# B&R Automation Studio project NAELD004C00R10L518F00 (part 35)

#### Act_Main.st
```iecst
(** 2020-03-16 **)
ACTION Act_Main:

	IF bModuleNotOK = FALSE THEN
		CASE eStat OF

			LifterActIdle:
				IF eStatus <> Idle THEN	//Reset Data
					//Private
					fbStop(bEn := FALSE);
					fbRstAxisErr(bEn := FALSE);
					fbJog(bEn := FALSE);
					fbMovRel(bEn := FALSE);
					fbMovAbs(bEn := FALSE);
					fbHoming(bEn := FALSE);
					fbPwrOff(bEn := FALSE);
					fbPwrOn(bEn := FALSE);
					fbFullHm(bEn := FALSE);
					fbFullMovAbs(bEn := FALSE);
					fbFullMovRel(bEn := FALSE);
					fbSDOWrite(bEn := FALSE);
					fbTm(IN := FALSE);
					usiStep	:= 0;
					usiCount			:= 0;
					bNotInterruptible	:= FALSE;

					sStatTxt	:= a_sStatText[eStat];

				END_IF

				eStatus	:= Idle;

				IF EDGENEG(p_bManual) THEN
					fMotionCANRstCtrlWord(ADR(tyParamOutDriver));
				END_IF

			LifterActGoAPos:
				IF (eStatus = Idle OR eStatus = Busy) THEN

					eStatus	:= Busy;

					sStatTxt	:= a_sStatText[eStat];

					bNotInterruptible	:= TRUE;

					CASE usiStep OF
						0:	//Wait For Motion Parameter Update
							p_diMovePosInUM	:= p_diAPos;
							usiStep	:= 1;

						1:	//Check Position Difference
							IF tyParamOut.bPosDiff = TRUE THEN
								usiStep	:= 2;
							ELSE
								eStatus	:= Done;
							END_IF

						2:	//Move
							fbFullMovAbs.tyParamInDriver					:= tyParamInDriver;
							fbFullMovAbs.tyParamInMove.diPosInUM			:= p_diMovePosInUM;
							fbFullMovAbs.tyParamInMove.diDistInUM			:= p_diMoveDistInUM;
							fbFullMovAbs.tyParamInMove.diVelInUMPS			:= p_diMoveVelInUMPS;
							fbFullMovAbs.tyParamInMove.diAcc				:= p_diMoveAcc;
							fbFullMovAbs.tyParamInMove.diDec				:= p_diMoveDec;
							fbFullMovAbs.tyParamOut							:= tyParamOut;
							fbFullMovAbs(bEn := TRUE);

							IF fbFullMovAbs.udiStatus = 0 THEN
								eStatus	:= Done;
							ELSIF fbFullMovAbs.udiStatus < 65534 THEN
								eStatus		:= Error;

								IF fbFullMovAbs.udiStatus = 1401 THEN
									udiStatus	:= 10002;	//Power On Time Out While Going A Position
								ELSIF fbFullMovAbs.udiStatus = 1402 THEN
									udiStatus	:= 10003;	//Homing Time Out While Going A Position
								ELSIF fbFullMovAbs.udiStatus = 1403 THEN
									udiStatus	:= 10004;	//Move Absolute Time Out While Going A Position
								ELSIF fbFullMovAbs.udiStatus = 1405 THEN
									udiStatus	:= 10005;	//Stop Motion Time Out While Going A Position
								ELSIF fbFullMovAbs.udiStatus = 1408 THEN
									udiStatus	:= 10006;	//Axis Error Reset Failed While Going A Position
								ELSIF fbFullMovAbs.udiStatus = 1409 THEN
									udiStatus	:= 10007;	//Axis Error Occur In Move Absolute While Going A Position
								ELSIF fbFullMovAbs.udiStatus = 1411 THEN
									udiStatus	:= 10008;	//Axis Error Occur In Homing While Going A Position
								ELSIF fbFullMovAbs.udiStatus = 1412 THEN
									udiStatus	:= 10009;	//Homing Done But Home Flag Is Not Activated While Going A Position
								ELSIF fbFullMovAbs.udiStatus = 1413 THEN
									udiStatus	:= 10010;	//Forward Limit Activated In Homing While Going A Position
								ELSIF fbFullMovAbs.udiStatus = 1414 THEN
									udiStatus	:= 10011;	//Reverse Limit Activated In Homing While Going A Position
								ELSIF fbFullMovAbs.udiStatus = 1415 THEN
									udiStatus	:= 10012;	//Forward Limit Activated In Move Absolute While Going A Position
								ELSIF fbFullMovAbs.udiStatus = 1416 THEN
									udiStatus	:= 10013;	//Reverse Limit Activated In Move Absolute While Going A Position
								ELSE
									udiStatus	:= fbFullMovAbs.udiStatus;
								END_IF
							END_IF

					END_CASE

				END_IF

			LifterActGoBPos:
				IF (eStatus = Idle OR eStatus = Busy) THEN

					eStatus	:= Busy;

					sStatTxt	:= a_sStatText[eStat];

					bNotInterruptible	:= TRUE;

					CASE usiStep OF
						0:	//Wait For Motion Parameter Update
							p_diMovePosInUM	:= p_diBPos;
							usiStep	:= 1;

						1:	//Check Position Difference
							IF tyParamOut.bPosDiff = TRUE THEN
								usiStep	:= 2;
							ELSE
								eStatus	:= Done;
							END_IF

						2:	//Move
							fbFullMovAbs.tyParamInDriver					:= tyParamInDriver;
							fbFullMovAbs.tyParamInMove.diPosInUM			:= p_diMovePosInUM;
							fbFullMovAbs.tyParamInMove.diDistInUM			:= p_diMoveDistInUM;
							fbFullMovAbs.tyParamInMove.diVelInUMPS			:= p_diMoveVelInUMPS;
							fbFullMovAbs.tyParamInMove.diAcc				:= p_diMoveAcc;
							fbFullMovAbs.tyParamInMove.diDec				:= p_diMoveDec;
							fbFullMovAbs.tyParamOut							:= tyParamOut;
							fbFullMovAbs(bEn := TRUE);

							IF fbFullMovAbs.udiStatus = 0 THEN
								eStatus	:= Done;
							ELSIF fbFullMovAbs.udiStatus < 65534 THEN
								eStatus		:= Error;

								IF fbFullMovAbs.udiStatus = 1401 THEN
									udiStatus	:= 10029;	//Power On Time Out While Going B Position
								ELSIF fbFullMovAbs.udiStatus = 1402 THEN
									udiStatus	:= 10030;	//Homing Time Out While Going B Position
								ELSIF fbFullMovAbs.udiStatus = 1403 THEN
									udiStatus	:= 10031;	//Move Absolute Time Out While Going B Position
								ELSIF fbFullMovAbs.udiStatus = 1405 THEN
									udiStatus	:= 10032;	//Stop Motion Time Out While Going B Position
								ELSIF fbFullMovAbs.udiStatus = 1408 THEN
									udiStatus	:= 10033;	//Axis Error Reset Failed While Going B Position
								ELSIF fbFullMovAbs.udiStatus = 1409 THEN
									udiStatus	:= 10034;	//Axis Error Occur In Move Absolute While Going B Position
								ELSIF fbFullMovAbs.udiStatus = 1411 THEN
									udiStatus	:= 10035;	//Axis Error Occur In Homing While Going B Position
								ELSIF fbFullMovAbs.udiStatus = 1412 THEN
									udiStatus	:= 10036;	//Homing Done But Home Flag Is Not Activated While Going B Position
								ELSIF fbFullMovAbs.udiStatus = 1413 THEN
									udiStatus	:= 10037;	//Forward Limit Activated In Homing While Going B Position
								ELSIF fbFullMovAbs.udiStatus = 1414 THEN
									udiStatus	:= 10038;	//Reverse Limit Activated In Homing While Going B Position
								ELSIF fbFullMovAbs.udiStatus = 1415 THEN
									udiStatus	:= 10039;	//Forward Limit Activated In Move Absolute While Going B Position
								ELSIF fbFullMovAbs.udiStatus = 1416 THEN
									udiStatus	:= 10040;	//Reverse Limit Activated In Move Absolute While Going B Position
								ELSE
									udiStatus	:= fbFullMovAbs.udiStatus;
								END_IF
							END_IF

					END_CASE

				END_IF

			LifterActGoCPos:
				IF (eStatus = Idle OR eStatus = Busy) THEN

					eStatus	:= Busy;

					sStatTxt	:= a_sStatText[eStat];

					bNotInterruptible	:= TRUE;

					CASE usiStep OF
						0:	//Wait For Motion Parameter Update
							p_diMovePosInUM	:= p_diCPos;
							usiStep	:= 1;

						1:	//Check Position Difference
							IF tyParamOut.bPosDiff = TRUE THEN
								usiStep	:= 2;
							ELSE
								eStatus	:= Done;
							END_IF

						2:	//Move
							fbFullMovAbs.tyParamInDriver					:= tyParamInDriver;
							fbFullMovAbs.tyParamInMove.diPosInUM			:= p_diMovePosInUM;
							fbFullMovAbs.tyParamInMove.diDistInUM			:= p_diMoveDistInUM;
							fbFullMovAbs.tyParamInMove.diVelInUMPS			:= p_diMoveVelInUMPS;
							fbFullMovAbs.tyParamInMove.diAcc				:= p_diMoveAcc;
							fbFullMovAbs.tyParamInMove.diDec				:= p_diMoveDec;
							fbFullMovAbs.tyParamOut							:= tyParamOut;
							fbFullMovAbs(bEn := TRUE);

							IF fbFullMovAbs.udiStatus = 0 THEN
								eStatus	:= Done;
							ELSIF fbFullMovAbs.udiStatus < 65534 THEN
								eStatus		:= Error;

								IF fbFullMovAbs.udiStatus = 1401 THEN
									udiStatus	:= 10078;	//Power On Time Out While Going C Position
								ELSIF fbFullMovAbs.udiStatus = 1402 THEN
									udiStatus	:= 10079;	//Homing Time Out While Going C Position
								ELSIF fbFullMovAbs.udiStatus = 1403 THEN
									udiStatus	:= 10080;	//Move Absolute Time Out While Going C Position
								ELSIF fbFullMovAbs.udiStatus = 1405 THEN
									udiStatus	:= 10081;	//Stop Motion Time Out While Going C Position
								ELSIF fbFullMovAbs.udiStatus = 1408 THEN
									udiStatus	:= 10082;	//Axis Error Reset Failed While Going C Position
								ELSIF fbFullMovAbs.udiStatus = 1409 THEN
									udiStatus	:= 10083;	//Axis Error Occur In Move Absolute While Going C Position
								ELSIF fbFullMovAbs.udiStatus = 1411 THEN
									udiStatus	:= 10084;	//Axis Error Occur In Homing While Going C Position
								ELSIF fbFullMovAbs.udiStatus = 1412 THEN
									udiStatus	:= 10085;	//Homing Done But Home Flag Is Not Activated While Going C Position
								ELSIF fbFullMovAbs.udiStatus = 1413 THEN
									udiStatus	:= 10086;	//Forward Limit Activated In Homing While Going C Position
								ELSIF fbFullMovAbs.udiStatus = 1414 THEN
									udiStatus	:= 10087;	//Reverse Limit Activated In Homing While Going C Position
								ELSIF fbFullMovAbs.udiStatus = 1415 THEN
									udiStatus	:= 10088;	//Forward Limit Activated In Move Absolute While Going C Position
								ELSIF fbFullMovAbs.udiStatus = 1416 THEN
									udiStatus	:= 10089;	//Reverse Limit Activated In Move Absolute While Going C Position
								ELSE
									udiStatus	:= fbFullMovAbs.udiStatus;
								END_IF
							END_IF

					END_CASE

				END_IF

			LifterActGoDPos:
				IF (eStatus = Idle OR eStatus = Busy) THEN

					eStatus	:= Busy;

					sStatTxt	:= a_sStatText[eStat];

					bNotInterruptible	:= TRUE;

					CASE usiStep OF
						0:	//Wait For Motion Parameter Update
							p_diMovePosInUM	:= p_diDPos;
							usiStep	:= 1;

						1:	//Check Position Difference
							IF tyParamOut.bPosDiff = TRUE THEN
								usiStep	:= 2;
							ELSE
								eStatus	:= Done;
							END_IF

						2:	//Move
							fbFullMovAbs.tyParamInDriver					:= tyParamInDriver;
							fbFullMovAbs.tyParamInMove.diPosInUM			:= p_diMovePosInUM;
							fbFullMovAbs.tyParamInMove.diDistInUM			:= p_diMoveDistInUM;
							fbFullMovAbs.tyParamInMove.diVelInUMPS			:= p_diMoveVelInUMPS;
							fbFullMovAbs.tyParamInMove.diAcc				:= p_diMoveAcc;
							fbFullMovAbs.tyParamInMove.diDec				:= p_diMoveDec;
							fbFullMovAbs.tyParamOut							:= tyParamOut;
							fbFullMovAbs(bEn := TRUE);

							IF fbFullMovAbs.udiStatus = 0 THEN
								eStatus	:= Done;
							ELSIF fbFullMovAbs.udiStatus < 65534 THEN
								eStatus		:= Error;

								IF fbFullMovAbs.udiStatus = 1401 THEN
									udiStatus	:= 10090;	//Power On Time Out While Going D Position
								ELSIF fbFullMovAbs.udiStatus = 1402 THEN
									udiStatus	:= 10091;	//Homing Time Out While Going D Position
								ELSIF fbFullMovAbs.udiStatus = 1403 THEN
									udiStatus	:= 10092;	//Move Absolute Time Out While Going D Position
								ELSIF fbFullMovAbs.udiStatus = 1405 THEN
									udiStatus	:= 10093;	//Stop Motion Time Out While Going D Position
								ELSIF fbFullMovAbs.udiStatus = 1408 THEN
									udiStatus	:= 10094;	//Axis Error Reset Failed While Going D Position
								ELSIF fbFullMovAbs.udiStatus = 1409 THEN
									udiStatus	:= 10095;	//Axis Error Occur In Move Absolute While Going D Position
								ELSIF fbFullMovAbs.udiStatus = 1411 THEN
									udiStatus	:= 10096;	//Axis Error Occur In Homing While Going D Position
								ELSIF fbFullMovAbs.udiStatus = 1412 THEN
									udiStatus	:= 10097;	//Homing Done But Home Flag Is Not Activated While Going D Position
								ELSIF fbFullMovAbs.udiStatus = 1413 THEN
									udiStatus	:= 10098;	//Forward Limit Activated In Homing While Going D Position
								ELSIF fbFullMovAbs.udiStatus = 1414 THEN
									udiStatus	:= 10099;	//Reverse Limit Activated In Homing While Going D Position
								ELSIF fbFullMovAbs.udiStatus = 1415 THEN
									udiStatus	:= 10100;	//Forward Limit Activated In Move Absolute While Going D Position
								ELSIF fbFullMovAbs.udiStatus = 1416 THEN
									udiStatus	:= 10101;	//Reverse Limit Activated In Move Absolute While Going D Position
								ELSE
									udiStatus	:= fbFullMovAbs.udiStatus;
								END_IF
							END_IF

					END_CASE

				END_IF

			LifterActGoEPos:
				IF (eStatus = Idle OR eStatus = Busy) THEN

					eStatus	:= Busy;

					sStatTxt	:= a_sStatText[eStat];

					bNotInterruptible	:= TRUE;

					CASE usiStep OF
						0:	//Wait For Motion Parameter Update
							p_diMovePosInUM	:= p_diEPos;
							usiStep	:= 1;

						1:	//Check Position Difference
							IF tyParamOut.bPosDiff = TRUE THEN
								usiStep	:= 2;
							ELSE
								eStatus	:= Done;
							END_IF

						2:	//Move
							fbFullMovAbs.tyParamInDriver					:= tyParamInDriver;
							fbFullMovAbs.tyParamInMove.diPosInUM			:= p_diMovePosInUM;
							fbFullMovAbs.tyParamInMove.diDistInUM			:= p_diMoveDistInUM;
							fbFullMovAbs.tyParamInMove.diVelInUMPS			:= p_diMoveVelInUMPS;
							fbFullMovAbs.tyParamInMove.diAcc				:= p_diMoveAcc;
							fbFullMovAbs.tyParamInMove.diDec				:= p_diMoveDec;
							fbFullMovAbs.tyParamOut							:= tyParamOut;
							fbFullMovAbs(bEn := TRUE);

							IF fbFullMovAbs.udiStatus = 0 THEN
								eStatus	:= Done;
							ELSIF fbFullMovAbs.udiStatus < 65534 THEN
								eStatus		:= Error;

								IF fbFullMovAbs.udiStatus = 1401 THEN
									udiStatus	:= 10102;	//Power On Time Out While Going E Position
								ELSIF fbFullMovAbs.udiStatus = 1402 THEN
									udiStatus	:= 10103;	//Homing Time Out While Going E Position
								ELSIF fbFullMovAbs.udiStatus = 1403 THEN
									udiStatus	:= 10104;	//Move Absolute Time Out While Going E Position
								ELSIF fbFullMovAbs.udiStatus = 1405 THEN
									udiStatus	:= 10105;	//Stop Motion Time Out While Going E Position
								ELSIF fbFullMovAbs.udiStatus = 1408 THEN
									udiStatus	:= 10106;	//Axis Error Reset Failed While Going E Position
								ELSIF fbFullMovAbs.udiStatus = 1409 THEN
									udiStatus	:= 10107;	//Axis Error Occur In Move Absolute While Going E Position
								ELSIF fbFullMovAbs.udiStatus = 1411 THEN
									udiStatus	:= 10108;	//Axis Error Occur In Homing While Going E Position
								ELSIF fbFullMovAbs.udiStatus = 1412 THEN
									udiStatus	:= 10109;	//Homing Done But Home Flag Is Not Activated While Going E Position
								ELSIF fbFullMovAbs.udiStatus = 1413 THEN
									udiStatus	:= 10110;	//Forward Limit Activated In Homing While Going E Position
								ELSIF fbFullMovAbs.udiStatus = 1414 THEN
									udiStatus	:= 10111;	//Reverse Limit Activated In Homing While Going E Position
								ELSIF fbFullMovAbs.udiStatus = 1415 THEN
									udiStatus	:= 10112;	//Forward Limit Activated In Move Absolute While Going E Position
								ELSIF fbFullMovAbs.udiStatus = 1416 THEN
									udiStatus	:= 10113;	//Reverse Limit Activated In Move Absolute While Going E Position
								ELSE
									udiStatus	:= fbFullMovAbs.udiStatus;
								END_IF
							END_IF

					END_CASE

				END_IF

			LifterActGoFPos:
				IF (eStatus = Idle OR eStatus = Busy) THEN

					eStatus	:= Busy;

					sStatTxt	:= a_sStatText[eStat];

					bNotInterruptible	:= TRUE;

					CASE usiStep OF
						0:	//Wait For Motion Parameter Update
							p_diMovePosInUM	:= p_diFPos;
							usiStep	:= 1;

						1:	//Check Position Difference
							IF tyParamOut.bPosDiff = TRUE THEN
								usiStep	:= 2;
							ELSE
								eStatus	:= Done;
							END_IF

						2:	//Move
							fbFullMovAbs.tyParamInDriver					:= tyParamInDriver;
							fbFullMovAbs.tyParamInMove.diPosInUM			:= p_diMovePosInUM;
							fbFullMovAbs.tyParamInMove.diDistInUM			:= p_diMoveDistInUM;
							fbFullMovAbs.tyParamInMove.diVelInUMPS			:= p_diMoveVelInUMPS;
							fbFullMovAbs.tyParamInMove.diAcc				:= p_diMoveAcc;
							fbFullMovAbs.tyParamInMove.diDec				:= p_diMoveDec;
							fbFullMovAbs.tyParamOut							:= tyParamOut;
							fbFullMovAbs(bEn := TRUE);

							IF fbFullMovAbs.udiStatus = 0 THEN
								eStatus	:= Done;
							ELSIF fbFullMovAbs.udiStatus < 65534 THEN
								eStatus		:= Error;

								IF fbFullMovAbs.udiStatus = 1401 THEN
									udiStatus	:= 10114;	//Power On Time Out While Going F Position
								ELSIF fbFullMovAbs.udiStatus = 1402 THEN
									udiStatus	:= 10115;	//Homing Time Out While Going F Position
								ELSIF fbFullMovAbs.udiStatus = 1403 THEN
									udiStatus	:= 10116;	//Move Absolute Time Out While Going F Position
								ELSIF fbFullMovAbs.udiStatus = 1405 THEN
									udiStatus	:= 10117;	//Stop Motion Time Out While Going F Position
								ELSIF fbFullMovAbs.udiStatus = 1408 THEN
									udiStatus	:= 10118;	//Axis Error Reset Failed While Going F Position
								ELSIF fbFullMovAbs.udiStatus = 1409 THEN
									udiStatus	:= 10119;	//Axis Error Occur In Move Absolute While Going F Position
								ELSIF fbFullMovAbs.udiStatus = 1411 THEN
									udiStatus	:= 10120;	//Axis Error Occur In Homing While Going F Position
								ELSIF fbFullMovAbs.udiStatus = 1412 THEN
									udiStatus	:= 10121;	//Homing Done But Home Flag Is Not Activated While Going F Position
								ELSIF fbFullMovAbs.udiStatus = 1413 THEN
									udiStatus	:= 10122;	//Forward Limit Activated In Homing While Going F Position
								ELSIF fbFullMovAbs.udiStatus = 1414 THEN
									udiStatus	:= 10123;	//Reverse Limit Activated In Homing While Going F Position
								ELSIF fbFullMovAbs.udiStatus = 1415 THEN
									udiStatus	:= 10124;	//Forward Limit Activated In Move Absolute While Going F Position
								ELSIF fbFullMovAbs.udiStatus = 1416 THEN
									udiStatus	:= 10125;	//Reverse Limit Activated In Move Absolute While Going F Position
								ELSE
									udiStatus	:= fbFullMovAbs.udiStatus;
								END_IF
							END_IF

					END_CASE

				END_IF

			LifterActGoGPos:
				IF (eStatus = Idle OR eStatus = Busy) THEN

					eStatus	:= Busy;

					sStatTxt	:= a_sStatText[eStat];

					bNotInterruptible	:= TRUE;

					CASE usiStep OF
						0:	//Wait For Motion Parameter Update
							p_diMovePosInUM	:= p_diGPos;
							usiStep	:= 1;

						1:	//Check Position Difference
							IF tyParamOut.bPosDiff = TRUE THEN
								usiStep	:= 2;
							ELSE
								eStatus	:= Done;
							END_IF

						2:	//Move
							fbFullMovAbs.tyParamInDriver					:= tyParamInDriver;
							fbFullMovAbs.tyParamInMove.diPosInUM			:= p_diMovePosInUM;
							fbFullMovAbs.tyParamInMove.diDistInUM			:= p_diMoveDistInUM;
							fbFullMovAbs.tyParamInMove.diVelInUMPS			:= p_diMoveVelInUMPS;
							fbFullMovAbs.tyParamInMove.diAcc				:= p_diMoveAcc;
							fbFullMovAbs.tyParamInMove.diDec				:= p_diMoveDec;
							fbFullMovAbs.tyParamOut							:= tyParamOut;
							fbFullMovAbs(bEn := TRUE);

							IF fbFullMovAbs.udiStatus = 0 THEN
								eStatus	:= Done;
							ELSIF fbFullMovAbs.udiStatus < 65534 THEN
								eStatus		:= Error;

								IF fbFullMovAbs.udiStatus = 1401 THEN
									udiStatus	:= 10126;	//Power On Time Out While Going G Position
								ELSIF fbFullMovAbs.udiStatus = 1402 THEN
									udiStatus	:= 10127;	//Homing Time Out While Going G Position
								ELSIF fbFullMovAbs.udiStatus = 1403 THEN
									udiStatus	:= 10128;	//Move Absolute Time Out While Going G Position
								ELSIF fbFullMovAbs.udiStatus = 1405 THEN
									udiStatus	:= 10129;	//Stop Motion Time Out While Going G Position
								ELSIF fbFullMovAbs.udiStatus = 1408 THEN
									udiStatus	:= 10130;	//Axis Error Reset Failed While Going G Position
								ELSIF fbFullMovAbs.udiStatus = 1409 THEN
									udiStatus	:= 10131;	//Axis Error Occur In Move Absolute While Going G Position
								ELSIF fbFullMovAbs.udiStatus = 1411 THEN
									udiStatus	:= 10132;	//Axis Error Occur In Homing While Going G Position
								ELSIF fbFullMovAbs.udiStatus = 1412 THEN
									udiStatus	:= 10133;	//Homing Done But Home Flag Is Not Activated While Going G Position
								ELSIF fbFullMovAbs.udiStatus = 1413 THEN
									udiStatus	:= 10134;	//Forward Limit Activated In Homing While Going G Position
								ELSIF fbFullMovAbs.udiStatus = 1414 THEN
									udiStatus	:= 10135;	//Reverse Limit Activated In Homing While Going G Position
								ELSIF fbFullMovAbs.udiStatus = 1415 THEN
									udiStatus	:= 10136;	//Forward Limit Activated In Move Absolute While Going G Position
								ELSIF fbFullMovAbs.udiStatus = 1416 THEN
									udiStatus	:= 10137;	//Reverse Limit Activated In Move Absolute While Going G Position
								ELSE
									udiStatus	:= fbFullMovAbs.udiStatus;
								END_IF
							END_IF

					END_CASE

				END_IF

			LifterActGoHPos:
				IF (eStatus = Idle OR eStatus = Busy) THEN

					eStatus	:= Busy;

					sStatTxt	:= a_sStatText[eStat];

					bNotInterruptible	:= TRUE;

					CASE usiStep OF
						0:	//Wait For Motion Parameter Update
							p_diMovePosInUM	:= p_diHPos;
							usiStep	:= 1;

						1:	//Check Position Difference
							IF tyParamOut.bPosDiff = TRUE THEN
								usiStep	:= 2;
							ELSE
								eStatus	:= Done;
							END_IF

						2:	//Move
							fbFullMovAbs.tyParamInDriver					:= tyParamInDriver;
							fbFullMovAbs.tyParamInMove.diPosInUM			:= p_diMovePosInUM;
							fbFullMovAbs.tyParamInMove.diDistInUM			:= p_diMoveDistInUM;
							fbFullMovAbs.tyParamInMove.diVelInUMPS			:= p_diMoveVelInUMPS;
							fbFullMovAbs.tyParamInMove.diAcc				:= p_diMoveAcc;
							fbFullMovAbs.tyParamInMove.diDec				:= p_diMoveDec;
							fbFullMovAbs.tyParamOut							:= tyParamOut;
							fbFullMovAbs(bEn := TRUE);

							IF fbFullMovAbs.udiStatus = 0 THEN
								eStatus	:= Done;
							ELSIF fbFullMovAbs.udiStatus < 65534 THEN
								eStatus		:= Error;

								IF fbFullMovAbs.udiStatus = 1401 THEN
									udiStatus	:= 10138;	//Power On Time Out While Going H Position
								ELSIF fbFullMovAbs.udiStatus = 1402 THEN
									udiStatus	:= 10139;	//Homing Time Out While Going H Position
								ELSIF fbFullMovAbs.udiStatus = 1403 THEN
									udiStatus	:= 10140;	//Move Absolute Time Out While Going H Position
								ELSIF fbFullMovAbs.udiStatus = 1405 THEN
									udiStatus	:= 10141;	//Stop Motion Time Out While Going H Position
								ELSIF fbFullMovAbs.udiStatus = 1408 THEN
									udiStatus	:= 10142;	//Axis Error Reset Failed While Going H Position
								ELSIF fbFullMovAbs.udiStatus = 1409 THEN
									udiStatus	:= 10143;	//Axis Error Occur In Move Absolute While Going H Position
								ELSIF fbFullMovAbs.udiStatus = 1411 THEN
									udiStatus	:= 10144;	//Axis Error Occur In Homing While Going H Position
								ELSIF fbFullMovAbs.udiStatus = 1412 THEN
									udiStatus	:= 10145;	//Homing Done But Home Flag Is Not Activated While Going H Position
								ELSIF fbFullMovAbs.udiStatus = 1413 THEN
									udiStatus	:= 10146;	//Forward Limit Activated In Homing While Going H Position
								ELSIF fbFullMovAbs.udiStatus = 1414 THEN
									udiStatus	:= 10147;	//Reverse Limit Activated In Homing While Going H Position
								ELSIF fbFullMovAbs.udiStatus = 1415 THEN
									udiStatus	:= 10148;	//Forward Limit Activated In Move Absolute While Going H Position
								ELSIF fbFullMovAbs.udiStatus = 1416 THEN
									udiStatus	:= 10149;	//Reverse Limit Activated In Move Absolute While Going H Position
								ELSE
									udiStatus	:= fbFullMovAbs.udiStatus;
								END_IF
							END_IF

					END_CASE

				END_IF

			LifterActGoASltPos:
				IF (eStatus = Idle OR eStatus = Busy) THEN

					eStatus	:= Busy;

					sStatTxt	:= a_sStatText[eStat];

					bNotInterruptible	:= TRUE;

					CASE usiStep OF
						0:	//Wait For Motion Parameter Update
							p_diMovePosInUM	:= fLifterSltToPosInUMBtmMin(p_diGoASlt , p_diASltToSltDist , p_diASlt1Pos);
							usiStep	:= 1;

						1:	//Check Position Difference
							IF tyParamOut.bPosDiff = TRUE THEN
								usiStep	:= 2;
							ELSE
								eStatus	:= Done;
							END_IF

						2:	//Move
							fbFullMovAbs.tyParamInDriver					:= tyParamInDriver;
							fbFullMovAbs.tyParamInMove.diPosInUM			:= p_diMovePosInUM;
							fbFullMovAbs.tyParamInMove.diDistInUM			:= p_diMoveDistInUM;
							fbFullMovAbs.tyParamInMove.diVelInUMPS			:= p_diMoveVelInUMPS;
							fbFullMovAbs.tyParamInMove.diAcc				:= p_diMoveAcc;
							fbFullMovAbs.tyParamInMove.diDec				:= p_diMoveDec;
							fbFullMovAbs.tyParamOut							:= tyParamOut;
							fbFullMovAbs(bEn := TRUE);

							IF fbFullMovAbs.udiStatus = 0 THEN
								eStatus	:= Done;
							ELSIF fbFullMovAbs.udiStatus < 65534 THEN
								eStatus		:= Error;

								IF fbFullMovAbs.udiStatus = 1401 THEN
									udiStatus	:= 10041;	//Power On Time Out While Going New A Slot Position
								ELSIF fbFullMovAbs.udiStatus = 1402 THEN
									udiStatus	:= 10042;	//Homing Time Out While Going New A Slot Position
								ELSIF fbFullMovAbs.udiStatus = 1403 THEN
									udiStatus	:= 10043;	//Move Absolute Time Out While Going New A Slot Position
								ELSIF fbFullMovAbs.udiStatus = 1405 THEN
									udiStatus	:= 10044;	//Stop Motion Time Out While Going New A Slot Position
								ELSIF fbFullMovAbs.udiStatus = 1408 THEN
									udiStatus	:= 10045;	//Axis Error Reset Failed While Going New A Slot Position
								ELSIF fbFullMovAbs.udiStatus = 1409 THEN
									udiStatus	:= 10046;	//Axis Error Occur In Move Absolute While Going New A Slot Position
								ELSIF fbFullMovAbs.udiStatus = 1411 THEN
									udiStatus	:= 10047;	//Axis Error Occur In Homing While Going New A Slot Position
								ELSIF fbFullMovAbs.udiStatus = 1412 THEN
									udiStatus	:= 10048;	//Homing Done But Home Flag Is Not Activated While Going New A Slot Position
								ELSIF fbFullMovAbs.udiStatus = 1413 THEN
									udiStatus	:= 10049;	//Forward Limit Activated In Homing While Going New A Slot Position
								ELSIF fbFullMovAbs.udiStatus = 1414 THEN
									udiStatus	:= 10050;	//Reverse Limit Activated In Homing While Going New A Slot Position
								ELSIF fbFullMovAbs.udiStatus = 1415 THEN
									udiStatus	:= 10051;	//Forward Limit Activated In Move Absolute While Going New A Slot Position
								ELSIF fbFullMovAbs.udiStatus = 1416 THEN
									udiStatus	:= 10052;	//Reverse Limit Activated In Move Absolute While Going New A Slot Position
								ELSE
									udiStatus	:= fbFullMovAbs.udiStatus;
								END_IF
							END_IF

					END_CASE

				END_IF

			LifterActGoNxtASltPos:
				IF (eStatus = Idle OR eStatus = Busy) THEN

					eStatus	:= Busy;

					sStatTxt	:= a_sStatText[eStat];

					bNotInterruptible	:= TRUE;

					CASE usiStep OF
						0:	//Wait For Motion Parameter Update
							diExpectSlt		:= fLifterPosInUMToSltBtmMin(tyParamOut.diActualPosInUM , p_diASltToSltDist , p_diASlt1Pos);
							diExpectPosInUM	:= fLifterSltToPosInUMBtmMin(diExpectSlt , p_diASltToSltDist , p_diASlt1Pos);

							IF ABS(tyParamOut.diActualPosInUM - diExpectPosInUM) < 50 THEN
								p_diGoASlt		:= diExpectSlt + 1;
								p_diMovePosInUM	:= fLifterSltToPosInUMBtmMin(p_diGoASlt , p_diASltToSltDist , p_diASlt1Pos);

							ELSIF tyParamOut.diActualPosInUM > diExpectPosInUM THEN
								p_diGoASlt		:= diExpectSlt;
								p_diMovePosInUM	:= fLifterSltToPosInUMBtmMin(p_diGoASlt , p_diASltToSltDist , p_diASlt1Pos);

							ELSIF tyParamOut.diActualPosInUM < diExpectPosInUM THEN
								p_diGoASlt		:= diExpectSlt + 1;
								p_diMovePosInUM	:= fLifterSltToPosInUMBtmMin(p_diGoASlt , p_diASltToSltDist , p_diASlt1Pos);

							END_IF

							usiStep	:= 1;

						1:	//Check Position Difference
							IF tyParamOut.bPosDiff = TRUE THEN
								usiStep	:= 2;
							ELSE
								eStatus	:= Done;
							END_IF

						2:	//Move
							fbFullMovAbs.tyParamInDriver					:= tyParamInDriver;
							fbFullMovAbs.tyParamInMove.diPosInUM			:= p_diMovePosInUM;
							fbFullMovAbs.tyParamInMove.diDistInUM			:= p_diMoveDistInUM;
							fbFullMovAbs.tyParamInMove.diVelInUMPS			:= p_diMoveVelInUMPS;
							fbFullMovAbs.tyParamInMove.diAcc				:= p_diMoveAcc;
							fbFullMovAbs.tyParamInMove.diDec				:= p_diMoveDec;
							fbFullMovAbs.tyParamOut							:= tyParamOut;
							fbFullMovAbs(bEn := TRUE);

							IF fbFullMovAbs.udiStatus = 0 THEN
								eStatus	:= Done;
							ELSIF fbFullMovAbs.udiStatus < 65534 THEN
								eStatus		:= Error;

								IF fbFullMovAbs.udiStatus = 1401 THEN
									udiStatus	:= 10053;	//Power On Time Out While Going Next A Slot Position
								ELSIF fbFullMovAbs.udiStatus = 1402 THEN
									udiStatus	:= 10054;	//Homing Time Out While Going Next A Slot Position
								ELSIF fbFullMovAbs.udiStatus = 1403 THEN
									udiStatus	:= 10055;	//Move Absolute Time Out While Going Next A Slot Position
								ELSIF fbFullMovAbs.udiStatus = 1405 THEN
									udiStatus	:= 10056;	//Stop Motion Time Out While Going Next A Slot Position
								ELSIF fbFullMovAbs.udiStatus = 1408 THEN
									udiStatus	:= 10057;	//Axis Error Reset Failed While Going Next A Slot Position
								ELSIF fbFullMovAbs.udiStatus = 1409 THEN
									udiStatus	:= 10058;	//Axis Error Occur In Move Absolute While Going Next A Slot Position
								ELSIF fbFullMovAbs.udiStatus = 1411 THEN
									udiStatus	:= 10059;	//Axis Error Occur In Homing While Going Next A Slot Position
								ELSIF fbFullMovAbs.udiStatus = 1412 THEN
									udiStatus	:= 10060;	//Homing Done But Home Flag Is Not Activated While Going Next A Slot Position
								ELSIF fbFullMovAbs.udiStatus = 1413 THEN
									udiStatus	:= 10061;	//Forward Limit Activated In Homing While Going Next A Slot Position
								ELSIF fbFullMovAbs.udiStatus = 1414 THEN
									udiStatus	:= 10062;	//Reverse Limit Activated In Homing While Going Next A Slot Position
								ELSIF fbFullMovAbs.udiStatus = 1415 THEN
									udiStatus	:= 10063;	//Forward Limit Activated In Move Absolute While Going Next A Slot Position
								ELSIF fbFullMovAbs.udiStatus = 1416 THEN
									udiStatus	:= 10064;	//Reverse Limit Activated In Move Absolute While Going Next A Slot Position
								ELSE
									udiStatus	:= fbFullMovAbs.udiStatus;
								END_IF
							END_IF

					END_CASE

				END_IF

			LifterActGoPrevASltPos:
				IF (eStatus = Idle OR eStatus = Busy) THEN

					eStatus	:= Busy;

					sStatTxt	:= a_sStatText[eStat];

					bNotInterruptible	:= TRUE;

					CASE usiStep OF
						0:	//Wait For Motion Parameter Update
							diExpectSlt		:= fLifterPosInUMToSltBtmMin(tyParamOut.diActualPosInUM , p_diASltToSltDist , p_diASlt1Pos);
							diExpectPosInUM	:= fLifterSltToPosInUMBtmMin(diExpectSlt , p_diASltToSltDist , p_diASlt1Pos);

							IF ABS(tyParamOut.diActualPosInUM - diExpectPosInUM) < 50 THEN
								p_diGoASlt		:= diExpectSlt - 1;
								p_diMovePosInUM	:= fLifterSltToPosInUMBtmMin(p_diGoASlt , p_diASltToSltDist , p_diASlt1Pos);

							ELSIF tyParamOut.diActualPosInUM > diExpectPosInUM THEN
								p_diGoASlt		:= diExpectSlt - 1;
								p_diMovePosInUM	:= fLifterSltToPosInUMBtmMin(p_diGoASlt , p_diASltToSltDist , p_diASlt1Pos);

							ELSIF tyParamOut.diActualPosInUM < diExpectPosInUM THEN
								p_diGoASlt		:= diExpectSlt;
								p_diMovePosInUM	:= fLifterSltToPosInUMBtmMin(p_diGoASlt , p_diASltToSltDist , p_diASlt1Pos);

							END_IF

							usiStep	:= 1;

						1:	//Check Position Difference
							IF tyParamOut.bPosDiff = TRUE THEN
								usiStep	:= 2;
							ELSE
								eStatus	:= Done;
							END_IF

						2:	//Move
							fbFullMovAbs.tyParamInDriver					:= tyParamInDriver;
							fbFullMovAbs.tyParamInMove.diPosInUM			:= p_diMovePosInUM;
							fbFullMovAbs.tyParamInMove.diDistInUM			:= p_diMoveDistInUM;
							fbFullMovAbs.tyParamInMove.diVelInUMPS			:= p_diMoveVelInUMPS;
							fbFullMovAbs.tyParamInMove.diAcc				:= p_diMoveAcc;
							fbFullMovAbs.tyParamInMove.diDec				:= p_diMoveDec;
							fbFullMovAbs.tyParamOut							:= tyParamOut;
							fbFullMovAbs(bEn := TRUE);

							IF fbFullMovAbs.udiStatus = 0 THEN
								eStatus	:= Done;
							ELSIF fbFullMovAbs.udiStatus < 65534 THEN
								eStatus		:= Error;

								IF fbFullMovAbs.udiStatus = 1401 THEN
									udiStatus	:= 10065;	//Power On Time Out While Going Previous A Slot Position
								ELSIF fbFullMovAbs.udiStatus = 1402 THEN
									udiStatus	:= 10066;	//Homing Time Out While Going Previous A Slot Position
								ELSIF fbFullMovAbs.udiStatus = 1403 THEN
									udiStatus	:= 10067;	//Move Absolute Time Out While Going Previous A Slot Position
								ELSIF fbFullMovAbs.udiStatus = 1405 THEN
									udiStatus	:= 10068;	//Stop Motion Time Out While Going Previous A Slot Position
								ELSIF fbFullMovAbs.udiStatus = 1408 THEN
									udiStatus	:= 10069;	//Axis Error Reset Failed While Going Previous A Slot Position
								ELSIF fbFullMovAbs.udiStatus = 1409 THEN
									udiStatus	:= 10070;	//Axis Error Occur In Move Absolute While Going Previous A Slot Position
								ELSIF fbFullMovAbs.udiStatus = 1411 THEN
									udiStatus	:= 10071;	//Axis Error Occur In Homing While Going Previous A Slot Position
								ELSIF fbFullMovAbs.udiStatus = 1412 THEN
									udiStatus	:= 10072;	//Homing Done But Home Flag Is Not Activated While Going Previous A Slot Position
								ELSIF fbFullMovAbs.udiStatus = 1413 THEN
									udiStatus	:= 10073;	//Forward Limit Activated In Homing While Going Previous A Slot Position
								ELSIF fbFullMovAbs.udiStatus = 1414 THEN
									udiStatus	:= 10074;	//Reverse Limit Activated In Homing While Going Previous A Slot Position
								ELSIF fbFullMovAbs.udiStatus = 1415 THEN
									udiStatus	:= 10075;	//Forward Limit Activated In Move Absolute While Going Previous A Slot Position
								ELSIF fbFullMovAbs.udiStatus = 1416 THEN
									udiStatus	:= 10076;	//Reverse Limit Activated In Move Absolute While Going Previous A Slot Position
								ELSE
									udiStatus	:= fbFullMovAbs.udiStatus;
								END_IF
							END_IF

					END_CASE

				END_IF

			LifterActGoBSltPos:
				IF (eStatus = Idle OR eStatus = Busy) THEN

					eStatus	:= Busy;

					sStatTxt	:= a_sStatText[eStat];

					bNotInterruptible	:= TRUE;

					CASE usiStep OF
						0:	//Wait For Motion Parameter Update
							p_diMovePosInUM	:= fLifterSltToPosInUMBtmMin(p_diGoBSlt , p_diBSltToSltDist , p_diBSlt1Pos);
							usiStep	:= 1;

						1:	//Check Position Difference
							IF tyParamOut.bPosDiff = TRUE THEN
								usiStep	:= 2;
							ELSE
								eStatus	:= Done;
							END_IF

						2:	//Move
							fbFullMovAbs.tyParamInDriver					:= tyParamInDriver;
							fbFullMovAbs.tyParamInMove.diPosInUM			:= p_diMovePosInUM;
							fbFullMovAbs.tyParamInMove.diDistInUM			:= p_diMoveDistInUM;
							fbFullMovAbs.tyParamInMove.diVelInUMPS			:= p_diMoveVelInUMPS;
							fbFullMovAbs.tyParamInMove.diAcc				:= p_diMoveAcc;
							fbFullMovAbs.tyParamInMove.diDec				:= p_diMoveDec;
							fbFullMovAbs.tyParamOut							:= tyParamOut;
							fbFullMovAbs(bEn := TRUE);

							IF fbFullMovAbs.udiStatus = 0 THEN
								eStatus	:= Done;
							ELSIF fbFullMovAbs.udiStatus < 65534 THEN
								eStatus		:= Error;

								IF fbFullMovAbs.udiStatus = 1401 THEN
									udiStatus	:= 10150;	//Power On Time Out While Going New B Slot Position
								ELSIF fbFullMovAbs.udiStatus = 1402 THEN
									udiStatus	:= 10151;	//Homing Time Out While Going New B Slot Position
								ELSIF fbFullMovAbs.udiStatus = 1403 THEN
									udiStatus	:= 10152;	//Move Absolute Time Out While Going New B Slot Position
								ELSIF fbFullMovAbs.udiStatus = 1405 THEN
									udiStatus	:= 10153;	//Stop Motion Time Out While Going New B Slot Position
								ELSIF fbFullMovAbs.udiStatus = 1408 THEN
									udiStatus	:= 10154;	//Axis Error Reset Failed While Going New B Slot Position
								ELSIF fbFullMovAbs.udiStatus = 1409 THEN
									udiStatus	:= 10155;	//Axis Error Occur In Move Absolute While Going New B Slot Position
								ELSIF fbFullMovAbs.udiStatus = 1411 THEN
									udiStatus	:= 10156;	//Axis Error Occur In Homing While Going New B Slot Position
								ELSIF fbFullMovAbs.udiStatus = 1412 THEN
									udiStatus	:= 10157;	//Homing Done But Home Flag Is Not Activated While Going New B Slot Position
								ELSIF fbFullMovAbs.udiStatus = 1413 THEN
									udiStatus	:= 10158;	//Forward Limit Activated In Homing While Going New B Slot Position
								ELSIF fbFullMovAbs.udiStatus = 1414 THEN
									udiStatus	:= 10159;	//Reverse Limit Activated In Homing While Going New B Slot Position
								ELSIF fbFullMovAbs.udiStatus = 1415 THEN
									udiStatus	:= 10160;	//Forward Limit Activated In Move Absolute While Going New B Slot Position
								ELSIF fbFullMovAbs.udiStatus = 1416 THEN
									udiStatus	:= 10161;	//Reverse Limit Activated In Move Absolute While Going New B Slot Position
								ELSE
									udiStatus	:= fbFullMovAbs.udiStatus;
								END_IF
							END_IF

					END_CASE

				END_IF

			LifterActGoNxtBSltPos:
				IF (eStatus = Idle OR eStatus = Busy) THEN

					eStatus	:= Busy;

					sStatTxt	:= a_sStatText[eStat];

					bNotInterruptible	:= TRUE;

					CASE usiStep OF
						0:	//Wait For Motion Parameter Update
							diExpectSlt		:= fLifterPosInUMToSltBtmMin(tyParamOut.diActualPosInUM , p_diBSltToSltDist , p_diBSlt1Pos);
							diExpectPosInUM	:= fLifterSltToPosInUMBtmMin(diExpectSlt , p_diBSltToSltDist , p_diBSlt1Pos);

							IF ABS(tyParamOut.diActualPosInUM - diExpectPosInUM) < 50 THEN
								p_diGoBSlt		:= diExpectSlt + 1;
								p_diMovePosInUM	:= fLifterSltToPosInUMBtmMin(p_diGoBSlt , p_diBSltToSltDist , p_diBSlt1Pos);

							ELSIF tyParamOut.diActualPosInUM > diExpectPosInUM THEN
								p_diGoBSlt		:= diExpectSlt;
								p_diMovePosInUM	:= fLifterSltToPosInUMBtmMin(p_diGoBSlt , p_diBSltToSltDist , p_diBSlt1Pos);

							ELSIF tyParamOut.diActualPosInUM < diExpectPosInUM THEN
								p_diGoBSlt		:= diExpectSlt + 1;
								p_diMovePosInUM	:= fLifterSltToPosInUMBtmMin(p_diGoBSlt , p_diBSltToSltDist , p_diBSlt1Pos);

							END_IF

							usiStep	:= 1;

						1:	//Check Position Difference
							IF tyParamOut.bPosDiff = TRUE THEN
								usiStep	:= 2;
							ELSE
								eStatus	:= Done;
							END_IF

						2:	//Move
							fbFullMovAbs.tyParamInDriver					:= tyParamInDriver;
							fbFullMovAbs.tyParamInMove.diPosInUM			:= p_diMovePosInUM;
							fbFullMovAbs.tyParamInMove.diDistInUM			:= p_diMoveDistInUM;
							fbFullMovAbs.tyParamInMove.diVelInUMPS			:= p_diMoveVelInUMPS;
							fbFullMovAbs.tyParamInMove.diAcc				:= p_diMoveAcc;
							fbFullMovAbs.tyParamInMove.diDec				:= p_diMoveDec;
							fbFullMovAbs.tyParamOut							:= tyParamOut;
							fbFullMovAbs(bEn := TRUE);

							IF fbFullMovAbs.udiStatus = 0 THEN
								eStatus	:= Done;
							ELSIF fbFullMovAbs.udiStatus < 65534 THEN
								eStatus		:= Error;

								IF fbFullMovAbs.udiStatus = 1401 THEN
									udiStatus	:= 10162;	//Power On Time Out While Going Next B Slot Position
								ELSIF fbFullMovAbs.udiStatus = 1402 THEN
									udiStatus	:= 10163;	//Homing Time Out While Going Next B Slot Position
								ELSIF fbFullMovAbs.udiStatus = 1403 THEN
									udiStatus	:= 10164;	//Move Absolute Time Out While Going Next B Slot Position
								ELSIF fbFullMovAbs.udiStatus = 1405 THEN
									udiStatus	:= 10165;	//Stop Motion Time Out While Going Next B Slot Position
								ELSIF fbFullMovAbs.udiStatus = 1408 THEN
									udiStatus	:= 10166;	//Axis Error Reset Failed While Going Next B Slot Position
								ELSIF fbFullMovAbs.udiStatus = 1409 THEN
									udiStatus	:= 10167;	//Axis Error Occur In Move Absolute While Going Next B Slot Position
								ELSIF fbFullMovAbs.udiStatus = 1411 THEN
									udiStatus	:= 10168;	//Axis Error Occur In Homing While Going Next B Slot Position
								ELSIF fbFullMovAbs.udiStatus = 1412 THEN
									udiStatus	:= 10169;	//Homing Done But Home Flag Is Not Activated While Going Next B Slot Position
								ELSIF fbFullMovAbs.udiStatus = 1413 THEN
									udiStatus	:= 10170;	//Forward Limit Activated In Homing While Going Next B Slot Position
								ELSIF fbFullMovAbs.udiStatus = 1414 THEN
									udiStatus	:= 10171;	//Reverse Limit Activated In Homing While Going Next B Slot Position
								ELSIF fbFullMovAbs.udiStatus = 1415 THEN
									udiStatus	:= 10172;	//Forward Limit Activated In Move Absolute While Going Next B Slot Position
								ELSIF fbFullMovAbs.udiStatus = 1416 THEN
									udiStatus	:= 10173;	//Reverse Limit Activated In Move Absolute While Going Next B Slot Position
								ELSE
									udiStatus	:= fbFullMovAbs.udiStatus;
								END_IF
							END_IF

					END_CASE

				END_IF

			LifterActGoPrevBSltPos:
				IF (eStatus = Idle OR eStatus = Busy) THEN

					eStatus	:= Busy;

					sStatTxt	:= a_sStatText[eStat];

					bNotInterruptible	:= TRUE;

					CASE usiStep OF
						0:	//Wait For Motion Parameter Update
							diExpectSlt		:= fLifterPosInUMToSltBtmMin(tyParamOut.diActualPosInUM , p_diBSltToSltDist , p_diBSlt1Pos);
							diExpectPosInUM	:= fLifterSltToPosInUMBtmMin(diExpectSlt , p_diBSltToSltDist , p_diBSlt1Pos);

							IF ABS(tyParamOut.diActualPosInUM - diExpectPosInUM) < 50 THEN
								p_diGoBSlt		:= diExpectSlt - 1;
								p_diMovePosInUM	:= fLifterSltToPosInUMBtmMin(p_diGoBSlt , p_diBSltToSltDist , p_diBSlt1Pos);

							ELSIF tyParamOut.diActualPosInUM > diExpectPosInUM THEN
								p_diGoBSlt		:= diExpectSlt - 1;
								p_diMovePosInUM	:= fLifterSltToPosInUMBtmMin(p_diGoBSlt , p_diBSltToSltDist , p_diBSlt1Pos);

							ELSIF tyParamOut.diActualPosInUM < diExpectPosInUM THEN
								p_diGoBSlt		:= diExpectSlt;
								p_diMovePosInUM	:= fLifterSltToPosInUMBtmMin(p_diGoBSlt , p_diBSltToSltDist , p_diBSlt1Pos);

							END_IF

							usiStep	:= 1;

						1:	//Check Position Difference
							IF tyParamOut.bPosDiff = TRUE THEN
								usiStep	:= 2;
							ELSE
								eStatus	:= Done;
							END_IF

						2:	//Move
							fbFullMovAbs.tyParamInDriver					:= tyParamInDriver;
							fbFullMovAbs.tyParamInMove.diPosInUM			:= p_diMovePosInUM;
							fbFullMovAbs.tyParamInMove.diDistInUM			:= p_diMoveDistInUM;
							fbFullMovAbs.tyParamInMove.diVelInUMPS			:= p_diMoveVelInUMPS;
							fbFullMovAbs.tyParamInMove.diAcc				:= p_diMoveAcc;
							fbFullMovAbs.tyParamInMove.diDec				:= p_diMoveDec;
							fbFullMovAbs.tyParamOut							:= tyParamOut;
							fbFullMovAbs(bEn := TRUE);

							IF fbFullMovAbs.udiStatus = 0 THEN
								eStatus	:= Done;
							ELSIF fbFullMovAbs.udiStatus < 65534 THEN
								eStatus		:= Error;

								IF fbFullMovAbs.udiStatus = 1401 THEN
									udiStatus	:= 10174;	//Power On Time Out While Going Previous B Slot Position
								ELSIF fbFullMovAbs.udiStatus = 1402 THEN
									udiStatus	:= 10175;	//Homing Time Out While Going Previous B Slot Position
								ELSIF fbFullMovAbs.udiStatus = 1403 THEN
									udiStatus	:= 10176;	//Move Absolute Time Out While Going Previous B Slot Position
								ELSIF fbFullMovAbs.udiStatus = 1405 THEN
									udiStatus	:= 10177;	//Stop Motion Time Out While Going Previous B Slot Position
								ELSIF fbFullMovAbs.udiStatus = 1408 THEN
									udiStatus	:= 10178;	//Axis Error Reset Failed While Going Previous B Slot Position
								ELSIF fbFullMovAbs.udiStatus = 1409 THEN
									udiStatus	:= 10179;	//Axis Error Occur In Move Absolute While Going Previous B Slot Position
								ELSIF fbFullMovAbs.udiStatus = 1411 THEN
									udiStatus	:= 10180;	//Axis Error Occur In Homing While Going Previous B Slot Position
								ELSIF fbFullMovAbs.udiStatus = 1412 THEN
									udiStatus	:= 10181;	//Homing Done But Home Flag Is Not Activated While Going Previous B Slot Position
								ELSIF fbFullMovAbs.udiStatus = 1413 THEN
									udiStatus	:= 10182;	//Forward Limit Activated In Homing While Going Previous B Slot Position
								ELSIF fbFullMovAbs.udiStatus = 1414 THEN
									udiStatus	:= 10183;	//Reverse Limit Activated In Homing While Going Previous B Slot Position
								ELSIF fbFullMovAbs.udiStatus = 1415 THEN
									udiStatus	:= 10184;	//Forward Limit Activated In Move Absolute While Going Previous B Slot Position
								ELSIF fbFullMovAbs.udiStatus = 1416 THEN
									udiStatus	:= 10185;	//Reverse Limit Activated In Move Absolute While Going Previous B Slot Position
								ELSE
									udiStatus	:= fbFullMovAbs.udiStatus;
								END_IF
							END_IF

					END_CASE

				END_IF

			LifterActGoCSltPos:
				IF (eStatus = Idle OR eStatus = Busy) THEN

					eStatus	:= Busy;

					sStatTxt	:= a_sStatText[eStat];

					bNotInterruptible	:= TRUE;

					CASE usiStep OF
						0:	//Wait For Motion Parameter Update
							p_diMovePosInUM	:= fLifterSltToPosInUMBtmMin(p_diGoCSlt , p_diCSltToSltDist , p_diCSlt1Pos);
							usiStep	:= 1;

						1:	//Check Position Difference
							IF tyParamOut.bPosDiff = TRUE THEN
								usiStep	:= 2;
							ELSE
								eStatus	:= Done;
							END_IF

						2:	//Move
							fbFullMovAbs.tyParamInDriver					:= tyParamInDriver;
							fbFullMovAbs.tyParamInMove.diPosInUM			:= p_diMovePosInUM;
							fbFullMovAbs.tyParamInMove.diDistInUM			:= p_diMoveDistInUM;
							fbFullMovAbs.tyParamInMove.diVelInUMPS			:= p_diMoveVelInUMPS;
							fbFullMovAbs.tyParamInMove.diAcc				:= p_diMoveAcc;
							fbFullMovAbs.tyParamInMove.diDec				:= p_diMoveDec;
							fbFullMovAbs.tyParamOut							:= tyParamOut;
							fbFullMovAbs(bEn := TRUE);

							IF fbFullMovAbs.udiStatus = 0 THEN
								eStatus	:= Done;
							ELSIF fbFullMovAbs.udiStatus < 65534 THEN
								eStatus		:= Error;

								IF fbFullMovAbs.udiStatus = 1401 THEN
									udiStatus	:= 10186;	//Power On Time Out While Going New C Slot Position
								ELSIF fbFullMovAbs.udiStatus = 1402 THEN
									udiStatus	:= 10187;	//Homing Time Out While Going New C  Slot Position
								ELSIF fbFullMovAbs.udiStatus = 1403 THEN
									udiStatus	:= 10188;	//Move Absolute Time Out While Going New C  Slot Position
								ELSIF fbFullMovAbs.udiStatus = 1405 THEN
									udiStatus	:= 10189;	//Stop Motion Time Out While Going New C  Slot Position
								ELSIF fbFullMovAbs.udiStatus = 1408 THEN
									udiStatus	:= 10190;	//Axis Error Reset Failed While Going New C  Slot Position
								ELSIF fbFullMovAbs.udiStatus = 1409 THEN
									udiStatus	:= 10191;	//Axis Error Occur In Move Absolute While Going New C  Slot Position
								ELSIF fbFullMovAbs.udiStatus = 1411 THEN
									udiStatus	:= 10192;	//Axis Error Occur In Homing While Going New C  Slot Position
								ELSIF fbFullMovAbs.udiStatus = 1412 THEN
									udiStatus	:= 10193;	//Homing Done But Home Flag Is Not Activated While Going New C  Slot Position
								ELSIF fbFullMovAbs.udiStatus = 1413 THEN
									udiStatus	:= 10194;	//Forward Limit Activated In Homing While Going New C  Slot Position
								ELSIF fbFullMovAbs.udiStatus = 1414 THEN
									udiStatus	:= 10195;	//Reverse Limit Activated In Homing While Going New C  Slot Position
								ELSIF fbFullMovAbs.udiStatus = 1415 THEN
									udiStatus	:= 10196;	//Forward Limit Activated In Move Absolute While Going New C  Slot Position
								ELSIF fbFullMovAbs.udiStatus = 1416 THEN
									udiStatus	:= 10197;	//Reverse Limit Activated In Move Absolute While Going New C  Slot Position
								ELSE
									udiStatus	:= fbFullMovAbs.udiStatus;
								END_IF
							END_IF

					END_CASE

				END_IF

			LifterActGoNxtCSltPos:
				IF (eStatus = Idle OR eStatus = Busy) THEN

					eStatus	:= Busy;

					sStatTxt	:= a_sStatText[eStat];

					bNotInterruptible	:= TRUE;

					CASE usiStep OF
						0:	//Wait For Motion Parameter Update
							diExpectSlt		:= fLifterPosInUMToSltBtmMin(tyParamOut.diActualPosInUM , p_diCSltToSltDist , p_diCSlt1Pos);
							diExpectPosInUM	:= fLifterSltToPosInUMBtmMin(diExpectSlt , p_diCSltToSltDist , p_diCSlt1Pos);

							IF ABS(tyParamOut.diActualPosInUM - diExpectPosInUM) < 50 THEN
								p_diGoCSlt		:= diExpectSlt + 1;
								p_diMovePosInUM	:= fLifterSltToPosInUMBtmMin(p_diGoCSlt , p_diCSltToSltDist , p_diCSlt1Pos);

							ELSIF tyParamOut.diActualPosInUM > diExpectPosInUM THEN
								p_diGoCSlt		:= diExpectSlt;
								p_diMovePosInUM	:= fLifterSltToPosInUMBtmMin(p_diGoCSlt , p_diCSltToSltDist , p_diCSlt1Pos);

							ELSIF tyParamOut.diActualPosInUM < diExpectPosInUM THEN
								p_diGoCSlt		:= diExpectSlt + 1;
								p_diMovePosInUM	:= fLifterSltToPosInUMBtmMin(p_diGoCSlt , p_diCSltToSltDist , p_diCSlt1Pos);

							END_IF

							usiStep	:= 1;

						1:	//Check Position Difference
							IF tyParamOut.bPosDiff = TRUE THEN
								usiStep	:= 2;
							ELSE
								eStatus	:= Done;
							END_IF

						2:	//Move
							fbFullMovAbs.tyParamInDriver					:= tyParamInDriver;
							fbFullMovAbs.tyParamInMove.diPosInUM			:= p_diMovePosInUM;
							fbFullMovAbs.tyParamInMove.diDistInUM			:= p_diMoveDistInUM;
							fbFullMovAbs.tyParamInMove.diVelInUMPS			:= p_diMoveVelInUMPS;
							fbFullMovAbs.tyParamInMove.diAcc				:= p_diMoveAcc;
							fbFullMovAbs.tyParamInMove.diDec				:= p_diMoveDec;
							fbFullMovAbs.tyParamOut							:= tyParamOut;
							fbFullMovAbs(bEn := TRUE);

							IF fbFullMovAbs.udiStatus = 0 THEN
								eStatus	:= Done;
							ELSIF fbFullMovAbs.udiStatus < 65534 THEN
								eStatus		:= Error;

								IF fbFullMovAbs.udiStatus = 1401 THEN
									udiStatus	:= 10198;	//Power On Time Out While Going Next C Slot Position
								ELSIF fbFullMovAbs.udiStatus = 1402 THEN
									udiStatus	:= 10199;	//Homing Time Out While Going Next C Slot Position
								ELSIF fbFullMovAbs.udiStatus = 1403 THEN
									udiStatus	:= 10200;	//Move Absolute Time Out While Going Next C Slot Position
								ELSIF fbFullMovAbs.udiStatus = 1405 THEN
									udiStatus	:= 10201;	//Stop Motion Time Out While Going Next C Slot Position
								ELSIF fbFullMovAbs.udiStatus = 1408 THEN
									udiStatus	:= 10202;	//Axis Error Reset Failed While Going Next C Slot Position
								ELSIF fbFullMovAbs.udiStatus = 1409 THEN
									udiStatus	:= 10203;	//Axis Error Occur In Move Absolute While Going Next C Slot Position
								ELSIF fbFullMovAbs.udiStatus = 1411 THEN
									udiStatus	:= 10204;	//Axis Error Occur In Homing While Going Next C Slot Position
								ELSIF fbFullMovAbs.udiStatus = 1412 THEN
									udiStatus	:= 10205;	//Homing Done But Home Flag Is Not Activated While Going Next C Slot Position
								ELSIF fbFullMovAbs.udiStatus = 1413 THEN
									udiStatus	:= 10206;	//Forward Limit Activated In Homing While Going Next C Slot Position
								ELSIF fbFullMovAbs.udiStatus = 1414 THEN
									udiStatus	:= 10207;	//Reverse Limit Activated In Homing While Going Next C Slot Position
								ELSIF fbFullMovAbs.udiStatus = 1415 THEN
									udiStatus	:= 10208;	//Forward Limit Activated In Move Absolute While Going Next C Slot Position
								ELSIF fbFullMovAbs.udiStatus = 1416 THEN
									udiStatus	:= 10209;	//Reverse Limit Activated In Move Absolute While Going Next C Slot Position
								ELSE
									udiStatus	:= fbFullMovAbs.udiStatus;
								END_IF
							END_IF

					END_CASE

				END_IF

			LifterActGoPrevCSltPos:
				IF (eStatus = Idle OR eStatus = Busy) THEN

					eStatus	:= Busy;

					sStatTxt	:= a_sStatText[eStat];

					bNotInterruptible	:= TRUE;

					CASE usiStep OF
						0:	//Wait For Motion Parameter Update
							diExpectSlt		:= fLifterPosInUMToSltBtmMin(tyParamOut.diActualPosInUM , p_diCSltToSltDist , p_diCSlt1Pos);
							diExpectPosInUM	:= fLifterSltToPosInUMBtmMin(diExpectSlt , p_diCSltToSltDist , p_diCSlt1Pos);

							IF ABS(tyParamOut.diActualPosInUM - diExpectPosInUM) < 50 THEN
								p_diGoCSlt		:= diExpectSlt - 1;
								p_diMovePosInUM	:= fLifterSltToPosInUMBtmMin(p_diGoCSlt , p_diCSltToSltDist , p_diCSlt1Pos);

							ELSIF tyParamOut.diActualPosInUM > diExpectPosInUM THEN
								p_diGoCSlt		:= diExpectSlt - 1;
								p_diMovePosInUM	:= fLifterSltToPosInUMBtmMin(p_diGoCSlt , p_diCSltToSltDist , p_diCSlt1Pos);

							ELSIF tyParamOut.diActualPosInUM < diExpectPosInUM THEN
								p_diGoCSlt		:= diExpectSlt;
								p_diMovePosInUM	:= fLifterSltToPosInUMBtmMin(p_diGoCSlt , p_diCSltToSltDist , p_diCSlt1Pos);

							END_IF

							usiStep	:= 1;

						1:	//Check Position Difference
							IF tyParamOut.bPosDiff = TRUE THEN
								usiStep	:= 2;
							ELSE
								eStatus	:= Done;
							END_IF

						2:	//Move
							fbFullMovAbs.tyParamInDriver					:= tyParamInDriver;
							fbFullMovAbs.tyParamInMove.diPosInUM			:= p_diMovePosInUM;
							fbFullMovAbs.tyParamInMove.diDistInUM			:= p_diMoveDistInUM;
							fbFullMovAbs.tyParamInMove.diVelInUMPS			:= p_diMoveVelInUMPS;
							fbFullMovAbs.tyParamInMove.diAcc				:= p_diMoveAcc;
							fbFullMovAbs.tyParamInMove.diDec				:= p_diMoveDec;
							fbFullMovAbs.tyParamOut							:= tyParamOut;
							fbFullMovAbs(bEn := TRUE);

							IF fbFullMovAbs.udiStatus = 0 THEN
								eStatus	:= Done;
							ELSIF fbFullMovAbs.udiStatus < 65534 THEN
								eStatus		:= Error;

								IF fbFullMovAbs.udiStatus = 1401 THEN
									udiStatus	:= 10210;	//Power On Time Out While Going Previous C Slot Position
								ELSIF fbFullMovAbs.udiStatus = 1402 THEN
									udiStatus	:= 10211;	//Homing Time Out While Going Previous C Slot Position
								ELSIF fbFullMovAbs.udiStatus = 1403 THEN
									udiStatus	:= 10212;	//Move Absolute Time Out While Going Previous C Slot Position
								ELSIF fbFullMovAbs.udiStatus = 1405 THEN
									udiStatus	:= 10213;	//Stop Motion Time Out While Going Previous C Slot Position
								ELSIF fbFullMovAbs.udiStatus = 1408 THEN
									udiStatus	:= 10214;	//Axis Error Reset Failed While Going Previous C Slot Position
								ELSIF fbFullMovAbs.udiStatus = 1409 THEN
									udiStatus	:= 10215;	//Axis Error Occur In Move Absolute While Going Previous C Slot Position
								ELSIF fbFullMovAbs.udiStatus = 1411 THEN
									udiStatus	:= 10216;	//Axis Error Occur In Homing While Going Previous C Slot Position
								ELSIF fbFullMovAbs.udiStatus = 1412 THEN
									udiStatus	:= 10217;	//Homing Done But Home Flag Is Not Activated While Going Previous C Slot Position
								ELSIF fbFullMovAbs.udiStatus = 1413 THEN
									udiStatus	:= 10218;	//Forward Limit Activated In Homing While Going Previous C Slot Position
								ELSIF fbFullMovAbs.udiStatus = 1414 THEN
									udiStatus	:= 10219;	//Reverse Limit Activated In Homing While Going Previous C Slot Position
								ELSIF fbFullMovAbs.udiStatus = 1415 THEN
									udiStatus	:= 10220;	//Forward Limit Activated In Move Absolute While Going Previous C Slot Position
								ELSIF fbFullMovAbs.udiStatus = 1416 THEN
									udiStatus	:= 10221;	//Reverse Limit Activated In Move Absolute While Going Previous C Slot Position
								ELSE
									udiStatus	:= fbFullMovAbs.udiStatus;
								END_IF
							END_IF

					END_CASE

				END_IF

			LifterActGoDSltPos:
				IF (eStatus = Idle OR eStatus = Busy) THEN

					eStatus	:= Busy;

					sStatTxt	:= a_sStatText[eStat];

					bNotInterruptible	:= TRUE;

					CASE usiStep OF
						0:	//Wait For Motion Parameter Update
							p_diMovePosInUM	:= fLifterSltToPosInUMBtmMin(p_diGoDSlt , p_diDSltToSltDist , p_diDSlt1Pos);
							usiStep	:= 1;

						1:	//Check Position Difference
							IF tyParamOut.bPosDiff = TRUE THEN
								usiStep	:= 2;
							ELSE
								eStatus	:= Done;
							END_IF

						2:	//Move
							fbFullMovAbs.tyParamInDriver					:= tyParamInDriver;
							fbFullMovAbs.tyParamInMove.diPosInUM			:= p_diMovePosInUM;
							fbFullMovAbs.tyParamInMove.diDistInUM			:= p_diMoveDistInUM;
							fbFullMovAbs.tyParamInMove.diVelInUMPS			:= p_diMoveVelInUMPS;
							fbFullMovAbs.tyParamInMove.diAcc				:= p_diMoveAcc;
							fbFullMovAbs.tyParamInMove.diDec				:= p_diMoveDec;
							fbFullMovAbs.tyParamOut							:= tyParamOut;
							fbFullMovAbs(bEn := TRUE);

							IF fbFullMovAbs.udiStatus = 0 THEN
								eStatus	:= Done;
							ELSIF fbFullMovAbs.udiStatus < 65534 THEN
								eStatus		:= Error;

								IF fbFullMovAbs.udiStatus = 1401 THEN
									udiStatus	:= 10222;	//Power On Time Out While Going New D Slot Position
								ELSIF fbFullMovAbs.udiStatus = 1402 THEN
									udiStatus	:= 10223;	//Homing Time Out While Going New D Slot Position
								ELSIF fbFullMovAbs.udiStatus = 1403 THEN
									udiStatus	:= 10224;	//Move Absolute Time Out While Going New D Slot Position
								ELSIF fbFullMovAbs.udiStatus = 1405 THEN
									udiStatus	:= 10225;	//Stop Motion Time Out While Going New D Slot Position
								ELSIF fbFullMovAbs.udiStatus = 1408 THEN
									udiStatus	:= 10226;	//Axis Error Reset Failed While Going New D Slot Position
								ELSIF fbFullMovAbs.udiStatus = 1409 THEN
									udiStatus	:= 10227;	//Axis Error Occur In Move Absolute While Going New D Slot Position
								ELSIF fbFullMovAbs.udiStatus = 1411 THEN
									udiStatus	:= 10228;	//Axis Error Occur In Homing While Going New D Slot Position
								ELSIF fbFullMovAbs.udiStatus = 1412 THEN
									udiStatus	:= 10229;	//Homing Done But Home Flag Is Not Activated While Going New D Slot Position
								ELSIF fbFullMovAbs.udiStatus = 1413 THEN
									udiStatus	:= 10230;	//Forward Limit Activated In Homing While Going New D Slot Position
								ELSIF fbFullMovAbs.udiStatus = 1414 THEN
									udiStatus	:= 10231;	//Reverse Limit Activated In Homing While Going New D Slot Position
								ELSIF fbFullMovAbs.udiStatus = 1415 THEN
									udiStatus	:= 10232;	//Forward Limit Activated In Move Absolute While Going New D Slot Position
								ELSIF fbFullMovAbs.udiStatus = 1416 THEN
									udiStatus	:= 10233;	//Reverse Limit Activated In Move Absolute While Going New D Slot Position
								ELSE
									udiStatus	:= fbFullMovAbs.udiStatus;
								END_IF
							END_IF

					END_CASE

				END_IF

			LifterActGoNxtDSltPos:
				IF (eStatus = Idle OR eStatus = Busy) THEN

					eStatus	:= Busy;

					sStatTxt	:= a_sStatText[eStat];

					bNotInterruptible	:= TRUE;

					CASE usiStep OF
						0:	//Wait For Motion Parameter Update
							diExpectSlt		:= fLifterPosInUMToSltBtmMin(tyParamOut.diActualPosInUM , p_diDSltToSltDist , p_diDSlt1Pos);
							diExpectPosInUM	:= fLifterSltToPosInUMBtmMin(diExpectSlt , p_diDSltToSltDist , p_diDSlt1Pos);

							IF ABS(tyParamOut.diActualPosInUM - diExpectPosInUM) < 50 THEN
								p_diGoDSlt		:= diExpectSlt + 1;
								p_diMovePosInUM	:= fLifterSltToPosInUMBtmMin(p_diGoDSlt , p_diDSltToSltDist , p_diDSlt1Pos);

							ELSIF tyParamOut.diActualPosInUM > diExpectPosInUM THEN
								p_diGoDSlt		:= diExpectSlt;
								p_diMovePosInUM	:= fLifterSltToPosInUMBtmMin(p_diGoDSlt , p_diDSltToSltDist , p_diDSlt1Pos);

							ELSIF tyParamOut.diActualPosInUM < diExpectPosInUM THEN
								p_diGoDSlt		:= diExpectSlt + 1;
								p_diMovePosInUM	:= fLifterSltToPosInUMBtmMin(p_diGoDSlt , p_diDSltToSltDist , p_diDSlt1Pos);

							END_IF

							usiStep	:= 1;

						1:	//Check Position Difference
							IF tyParamOut.bPosDiff = TRUE THEN
								usiStep	:= 2;
							ELSE
								eStatus	:= Done;
							END_IF

						2:	//Move
							fbFullMovAbs.tyParamInDriver					:= tyParamInDriver;
							fbFullMovAbs.tyParamInMove.diPosInUM			:= p_diMovePosInUM;
							fbFullMovAbs.tyParamInMove.diDistInUM			:= p_diMoveDistInUM;
							fbFullMovAbs.tyParamInMove.diVelInUMPS			:= p_diMoveVelInUMPS;
							fbFullMovAbs.tyParamInMove.diAcc				:= p_diMoveAcc;
							fbFullMovAbs.tyParamInMove.diDec				:= p_diMoveDec;
							fbFullMovAbs.tyParamOut							:= tyParamOut;
							fbFullMovAbs(bEn := TRUE);

							IF fbFullMovAbs.udiStatus = 0 THEN
								eStatus	:= Done;
							ELSIF fbFullMovAbs.udiStatus < 65534 THEN
								eStatus		:= Error;

								IF fbFullMovAbs.udiStatus = 1401 THEN
									udiStatus	:= 10234;	//Power On Time Out While Going Next D Slot Position
								ELSIF fbFullMovAbs.udiStatus = 1402 THEN
									udiStatus	:= 10235;	//Homing Time Out While Going Next D Slot Position
								ELSIF fbFullMovAbs.udiStatus = 1403 THEN
									udiStatus	:= 10236;	//Move Absolute Time Out While Going Next D Slot Position
								ELSIF fbFullMovAbs.udiStatus = 1405 THEN
									udiStatus	:= 10237;	//Stop Motion Time Out While Going Next D Slot Position
								ELSIF fbFullMovAbs.udiStatus = 1408 THEN
									udiStatus	:= 10238;	//Axis Error Reset Failed While Going Next D Slot Position
								ELSIF fbFullMovAbs.udiStatus = 1409 THEN
									udiStatus	:= 10239;	//Axis Error Occur In Move Absolute While Going Next D Slot Position
								ELSIF fbFullMovAbs.udiStatus = 1411 THEN
									udiStatus	:= 10240;	//Axis Error Occur In Homing While Going Next D Slot Position
								ELSIF fbFullMovAbs.udiStatus = 1412 THEN
									udiStatus	:= 10241;	//Homing Done But Home Flag Is Not Activated While Going Next D Slot Position
								ELSIF fbFullMovAbs.udiStatus = 1413 THEN
									udiStatus	:= 10242;	//Forward Limit Activated In Homing While Going Next D Slot Position
								ELSIF fbFullMovAbs.udiStatus = 1414 THEN
									udiStatus	:= 10243;	//Reverse Limit Activated In Homing While Going Next D Slot Position
								ELSIF fbFullMovAbs.udiStatus = 1415 THEN
									udiStatus	:= 10244;	//Forward Limit Activated In Move Absolute While Going Next D Slot Position
								ELSIF fbFullMovAbs.udiStatus = 1416 THEN
									udiStatus	:= 10245;	//Reverse Limit Activated In Move Absolute While Going Next D Slot Position
								ELSE
									udiStatus	:= fbFullMovAbs.udiStatus;
								END_IF
							END_IF

					END_CASE

				END_IF

			LifterActGoPrevDSltPos:
				IF (eStatus = Idle OR eStatus = Busy) THEN

					eStatus	:= Busy;

					sStatTxt	:= a_sStatText[eStat];

					bNotInterruptible	:= TRUE;

					CASE usiStep OF
						0:	//Wait For Motion Parameter Update
							diExpectSlt		:= fLifterPosInUMToSltBtmMin(tyParamOut.diActualPosInUM , p_diDSltToSltDist , p_diDSlt1Pos);
							diExpectPosInUM	:= fLifterSltToPosInUMBtmMin(diExpectSlt , p_diDSltToSltDist , p_diDSlt1Pos);

							IF ABS(tyParamOut.diActualPosInUM - diExpectPosInUM) < 50 THEN
								p_diGoDSlt		:= diExpectSlt - 1;
								p_diMovePosInUM	:= fLifterSltToPosInUMBtmMin(p_diGoDSlt , p_diDSltToSltDist , p_diDSlt1Pos);

							ELSIF tyParamOut.diActualPosInUM > diExpectPosInUM THEN
								p_diGoDSlt		:= diExpectSlt - 1;
								p_diMovePosInUM	:= fLifterSltToPosInUMBtmMin(p_diGoDSlt , p_diDSltToSltDist , p_diDSlt1Pos);

							ELSIF tyParamOut.diActualPosInUM < diExpectPosInUM THEN
								p_diGoDSlt		:= diExpectSlt;
								p_diMovePosInUM	:= fLifterSltToPosInUMBtmMin(p_diGoDSlt , p_diDSltToSltDist , p_diDSlt1Pos);

							END_IF

							usiStep	:= 1;

						1:	//Check Position Difference
							IF tyParamOut.bPosDiff = TRUE THEN
								usiStep	:= 2;
							ELSE
								eStatus	:= Done;
							END_IF

						2:	//Move
							fbFullMovAbs.tyParamInDriver					:= tyParamInDriver;
							fbFullMovAbs.tyParamInMove.diPosInUM			:= p_diMovePosInUM;
							fbFullMovAbs.tyParamInMove.diDistInUM			:= p_diMoveDistInUM;
							fbFullMovAbs.tyParamInMove.diVelInUMPS			:= p_diMoveVelInUMPS;
							fbFullMovAbs.tyParamInMove.diAcc				:= p_diMoveAcc;
							fbFullMovAbs.tyParamInMove.diDec				:= p_diMoveDec;
							fbFullMovAbs.tyParamOut							:= tyParamOut;
							fbFullMovAbs(bEn := TRUE);

							IF fbFullMovAbs.udiStatus = 0 THEN
								eStatus	:= Done;
							ELSIF fbFullMovAbs.udiStatus < 65534 THEN
								eStatus		:= Error;

								IF fbFullMovAbs.udiStatus = 1401 THEN
									udiStatus	:= 10246;	//Power On Time Out While Going Previous D Slot Position
								ELSIF fbFullMovAbs.udiStatus = 1402 THEN
									udiStatus	:= 10247;	//Homing Time Out While Going Previous D Slot Position
								ELSIF fbFullMovAbs.udiStatus = 1403 THEN
									udiStatus	:= 10248;	//Move Absolute Time Out While Going Previous D Slot Position
								ELSIF fbFullMovAbs.udiStatus = 1405 THEN
									udiStatus	:= 10249;	//Stop Motion Time Out While Going Previous D Slot Position
								ELSIF fbFullMovAbs.udiStatus = 1408 THEN
									udiStatus	:= 10250;	//Axis Error Reset Failed While Going Previous D Slot Position
								ELSIF fbFullMovAbs.udiStatus = 1409 THEN
									udiStatus	:= 10251;	//Axis Error Occur In Move Absolute While Going Previous D Slot Position
								ELSIF fbFullMovAbs.udiStatus = 1411 THEN
									udiStatus	:= 10252;	//Axis Error Occur In Homing While Going Previous D Slot Position
								ELSIF fbFullMovAbs.udiStatus = 1412 THEN
									udiStatus	:= 10253;	//Homing Done But Home Flag Is Not Activated While Going Previous D Slot Position
								ELSIF fbFullMovAbs.udiStatus = 1413 THEN
									udiStatus	:= 10254;	//Forward Limit Activated In Homing While Going Previous D Slot Position
								ELSIF fbFullMovAbs.udiStatus = 1414 THEN
									udiStatus	:= 10255;	//Reverse Limit Activated In Homing While Going Previous D Slot Position
								ELSIF fbFullMovAbs.udiStatus = 1415 THEN
									udiStatus	:= 10256;	//Forward Limit Activated In Move Absolute While Going Previous D Slot Position
								ELSIF fbFullMovAbs.udiStatus = 1416 THEN
									udiStatus	:= 10257;	//Reverse Limit Activated In Move Absolute While Going Previous D Slot Position
								ELSE
									udiStatus	:= fbFullMovAbs.udiStatus;
								END_IF
							END_IF

					END_CASE

				END_IF

			LifterActFullHm:
				IF (eStatus = Idle OR eStatus = Busy) THEN

					eStatus	:= Busy;

					sStatTxt	:= a_sStatText[eStat];

					bNotInterruptible	:= TRUE;

					fbFullHm.tyParamInDriver	:= tyParamInDriver;
					fbFullHm.tyParamOut			:= tyParamOut;
					fbFullHm(bEn := TRUE);

					IF fbFullHm.udiStatus = 0 THEN
						eStatus	:= Done;
					ELSIF fbFullHm.udiStatus < 65534 THEN
						eStatus		:= Error;

						IF fbFullHm.udiStatus = 1401 THEN
							udiStatus	:= 10014;	//Power On Time Out While Full Homing
						ELSIF fbFullHm.udiStatus = 1402 THEN
							udiStatus	:= 10015;	//Homing Time Out While Full Homing
						ELSIF fbFullHm.udiStatus = 1405 THEN
							udiStatus	:= 10016;	//Stop Motion Time Out While Full Homing
						ELSIF fbFullHm.udiStatus = 1408 THEN
							udiStatus	:= 10017;	//Axis Error Reset Failed While Full Homing
						ELSIF fbFullHm.udiStatus = 1411 THEN
							udiStatus	:= 10018;	//Axis Error Occur In Homing While Full Homing
						ELSIF fbFullHm.udiStatus = 1412 THEN
							udiStatus	:= 10019;	//Homing Done But Home Flag Is Not Activated While Full Homing
						ELSIF fbFullHm.udiStatus = 1413 THEN
							udiStatus	:= 10020;	//Forward Limit Activated In Homing While Full Homing
						ELSIF fbFullHm.udiStatus = 1414 THEN
							udiStatus	:= 10021;	//Reverse Limit Activated In Homing While Full Homing
						ELSE
							udiStatus	:= fbFullHm.udiStatus;
						END_IF
					END_IF

				END_IF

			LifterActFullMovRel:
				IF (eStatus = Idle OR eStatus = Busy) THEN

					eStatus	:= Busy;

					sStatTxt	:= a_sStatText[eStat];

					bNotInterruptible	:= TRUE;

					fbFullMovRel.tyParamInDriver					:= tyParamInDriver;
					fbFullMovRel.tyParamInMove.diPosInUM			:= p_diMovePosInUM;
					fbFullMovRel.tyParamInMove.diDistInUM			:= p_diMoveDistInUM;
					fbFullMovRel.tyParamInMove.diVelInUMPS			:= p_diMoveVelInUMPS;
					fbFullMovRel.tyParamOut							:= tyParamOut;
					fbFullMovRel(bEn := TRUE);

					IF fbFullMovRel.udiStatus = 0 THEN
						eStatus	:= Done;
					ELSIF fbFullMovRel.udiStatus < 65534 THEN
						eStatus		:= Error;

						IF fbFullMovRel.udiStatus = 1401 THEN
							udiStatus	:= 10259;	//Power On Time Out While Full Moving Relative
						ELSIF fbFullMovRel.udiStatus = 1404 THEN
							udiStatus	:= 10260;	//Move Relative Time Out Full Moving Relative
						ELSIF fbFullMovRel.udiStatus = 1405 THEN
							udiStatus	:= 10261;	//Stop Motion Time Out While Full Moving Relative
						ELSIF fbFullMovRel.udiStatus = 1408 THEN
							udiStatus	:= 10262;	//Axis Error Reset Failed While Full Moving Relative
						ELSE
							udiStatus	:= fbFullMovRel.udiStatus;
						END_IF
					END_IF

				END_IF

			LifterActPwrOn:
				IF (eStatus = Idle OR eStatus = Busy) THEN

					eStatus	:= Busy;

					sStatTxt	:= a_sStatText[eStat];

					fbPwrOn.tyParamInDriver	:= tyParamInDriver;
					fbPwrOn(bEn := TRUE);

					IF fbPwrOn.udiStatus = 0 THEN
						eStatus	:= Done;
					ELSIF fbPwrOn.udiStatus < 65534 THEN
						eStatus		:= Error;

						IF fbPwrOn.udiStatus = 1401 THEN
							udiStatus	:= 10022;	//Power On Time Out
						ELSE
							udiStatus	:= fbPwrOn.udiStatus;
						END_IF
					END_IF

				END_IF

			LifterActPwrOff:
				IF (eStatus = Idle OR eStatus = Busy) THEN

					eStatus	:= Busy;

					sStatTxt	:= a_sStatText[eStat];

					fbPwrOff.tyParamInDriver	:= tyParamInDriver;
					fbPwrOff(bEn := TRUE);

					IF fbPwrOff.udiStatus = 0 THEN
						eStatus	:= Done;
					ELSIF fbPwrOff.udiStatus < 65534 THEN
						eStatus		:= Error;

						IF fbPwrOff.udiStatus = 1400 THEN
							udiStatus	:= 10023;	//Power Off Time Out
						ELSE
							udiStatus	:= fbPwrOff.udiStatus;
						END_IF
					END_IF

				END_IF

			LifterActHoming:
				IF (eStatus = Idle OR eStatus = Busy) THEN

					eStatus	:= Busy;

					sStatTxt	:= a_sStatText[eStat];

					bNotInterruptible	:= TRUE;

					fbHoming.tyParamInDriver	:= tyParamInDriver;
					fbHoming.tyParamOut			:= tyParamOut;
					fbHoming(bEn := TRUE);

					IF fbHoming.udiStatus = 0 THEN
						eStatus	:= Done;
					ELSIF fbHoming.udiStatus < 65534 THEN
						eStatus		:= Error;

						IF fbHoming.udiStatus = 1402 THEN
							udiStatus	:= 10024;	//Homing Time Out
						ELSIF fbHoming.udiStatus = 1411 THEN
							udiStatus	:= 10018;	//Axis Error Occur In Homing While Full Homing

						ELSIF fbHoming.udiStatus = 1413 THEN
							udiStatus	:= 10020;	//Forward Limit Activated In Homing While Full Homing
						ELSIF fbHoming.udiStatus = 1414 THEN
							udiStatus	:= 10021;	//Reverse Limit Activated In Homing While Full Homing
						ELSE
							udiStatus	:= fbHoming.udiStatus;
						END_IF
					END_IF

				END_IF

			LifterActMovAbs:
				IF (eStatus = Idle OR eStatus = Busy) THEN

					eStatus	:= Busy;

					sStatTxt	:= a_sStatText[eStat];

					bNotInterruptible	:= TRUE;

					fbMovAbs.tyParamInDriver					:= tyParamInDriver;
					fbMovAbs.tyParamInMove.diPosInUM			:= p_diMovePosInUM;
					fbMovAbs.tyParamInMove.diDistInUM			:= p_diMoveDistInUM;
					fbMovAbs.tyParamInMove.diVelInUMPS			:= p_diMoveVelInUMPS;
					fbFullMovAbs.tyParamInMove.diAcc				:= p_diMoveAcc;
					fbFullMovAbs.tyParamInMove.diDec				:= p_diMoveDec;
					fbMovAbs(bEn := TRUE);

					IF fbMovAbs.udiStatus = 0 THEN
						eStatus	:= Done;
					ELSIF fbMovAbs.udiStatus < 65534 THEN
						eStatus		:= Error;

						IF fbMovAbs.udiStatus = 1403 THEN
							udiStatus	:= 10025;	//Move Absolute Time Out
						ELSE
							udiStatus	:= fbMovAbs.udiStatus;
						END_IF
					END_IF

				END_IF

			LifterActMovRel:
				IF (eStatus = Idle OR eStatus = Busy) THEN

					eStatus	:= Busy;

					sStatTxt	:= a_sStatText[eStat];

					bNotInterruptible	:= TRUE;

					fbMovRel.tyParamInDriver					:= tyParamInDriver;
					fbMovRel.tyParamInMove.diPosInUM			:= p_diMovePosInUM;
					fbMovRel.tyParamInMove.diDistInUM			:= p_diMoveDistInUM;
					fbMovRel.tyParamInMove.diVelInUMPS			:= p_diMoveVelInUMPS;
					fbMovRel.tyParamInMove.diAcc				:= p_diMoveAcc;
					fbMovRel.tyParamInMove.diDec				:= p_diMoveDec;
					fbMovRel(bEn := TRUE);

					IF fbMovRel.udiStatus = 0 THEN
						eStatus	:= Done;
					ELSIF fbMovRel.udiStatus < 65534 THEN
						eStatus		:= Error;

						IF fbMovRel.udiStatus = 1404 THEN
							udiStatus	:= 10026;	//Move Relative Time Out
						ELSE
							udiStatus	:= fbMovRel.udiStatus;
						END_IF
					END_IF

				END_IF

			LifterActJogUp:
				IF (eStatus = Idle OR eStatus = Busy) THEN

					eStatus	:= Busy;

					sStatTxt	:= a_sStatText[eStat];

					fbJog.tyParamInDriver	:= tyParamInDriver;
					fbJog.tyParamInMove.diAcc		:= p_diMoveAcc;
					fbJog.tyParamInMove.diDec		:= p_diMoveDec;

					IF p_bDir = TRUE THEN
						fbJog.tyParamInJog.diVelInUMPS	:= p_diJogVelInUMPS * -1;
					ELSE
						fbJog.tyParamInJog.diVelInUMPS	:= p_diJogVelInUMPS;
					END_IF

					fbJog(bEn := TRUE);

					IF fbJog.udiStatus = 0 THEN
						bJogging	:= TRUE;
						eStatus		:= Done;
					ELSIF fbJog.udiStatus < 65534 THEN
						udiStatus	:= fbJog.udiStatus;
						eStatus		:= Error;
					END_IF

				END_IF

			LifterActJogDown:
				IF (eStatus = Idle OR eStatus = Busy) THEN

					eStatus	:= Busy;

					sStatTxt	:= a_sStatText[eStat];

					bNotInterruptible	:= TRUE;

					fbJog.tyParamInDriver	:= tyParamInDriver;
					fbJog.tyParamInMove.diAcc		:= p_diMoveAcc;
					fbJog.tyParamInMove.diDec		:= p_diMoveDec;

					IF p_bDir = TRUE THEN
						fbJog.tyParamInJog.diVelInUMPS	:= p_diJogVelInUMPS;
					ELSE
						fbJog.tyParamInJog.diVelInUMPS	:= p_diJogVelInUMPS * -1;
					END_IF

					fbJog(bEn := TRUE);

					IF fbJog.udiStatus = 0 THEN
						bJogging	:= TRUE;
						eStatus		:= Done;
					ELSIF fbJog.udiStatus < 65534 THEN
						udiStatus	:= fbJog.udiStatus;
						eStatus		:= Error;
					END_IF

				END_IF

			LifterActJogStop:
				IF (eStatus = Idle OR eStatus = Busy) THEN

					sStatTxt	:= a_sStatText[eStat];

					fMotionCANJogStop(ADR(tyParamOutDriver));
					bJogging	:= FALSE;

					eStatus	:= Done;

				END_IF

			LifterActRstAxisErr:
				IF (eStatus = Idle OR eStatus = Busy) THEN

					eStatus	:= Busy;

					sStatTxt	:= a_sStatText[eStat];

					fbRstAxisErr(bEn := TRUE);

					IF fbRstAxisErr.udiStatus = 0 THEN
						eStatus	:= Done;
					ELSIF fbRstAxisErr.udiStatus < 65534 THEN
						udiStatus	:= fbRstAxisErr.udiStatus;
						eStatus		:= Error;
					END_IF

				END_IF

			LifterActStop:
				IF (eStatus = Idle OR eStatus = Busy) THEN

					eStatus	:= Busy;

					sStatTxt	:= a_sStatText[eStat];

					fbStop.tyParamInDriver	:= tyParamInDriver;
					fbStop(bEn := TRUE);

					IF fbStop.udiStatus = 0 THEN
						bJogging	:= FALSE;
						eStatus		:= Done;
					ELSIF fbStop.udiStatus < 65534 THEN
						eStatus		:= Error;

						IF fbStop.udiStatus = 1405 THEN
							udiStatus	:= 10027;	//Stop Motion Time Out
						ELSE
							udiStatus	:= fbStop.udiStatus;
						END_IF
					END_IF

				END_IF
		END_CASE
ELSE
	CASE eStat OF
		LifterActSDOWrite:
			IF (eStatus = Idle OR eStatus = Busy) THEN

				eStatus	:= Busy;

				sStatTxt	:= a_sStatText[eStat];

				fbTm(IN := TRUE);

				IF fbTm.Q THEN

					fbSDOWrite.tyParamOut	:= tyParamOut;
					fbSDOWrite.tyTuning		:= p_tyTuning;
					fbSDOWrite(bEn := TRUE);

					IF fbSDOWrite.udiStatus = 0 THEN
						eStatus	:= Done;
					ELSIF fbSDOWrite.udiStatus < 65534 THEN
						fMotionCANRstCtrlWord(ADR(tyParamOutDriver));

						IF usiCount < 5 THEN
							fbTm(IN := FALSE);
							fbSDOWrite(bEn := FALSE);

							usiCount	:= usiCount + 1;
						ELSE
							eStatus		:= Error;

							IF fbSDOWrite.udiStatus = 1406 THEN
								udiStatus	:= 10028;	//SDO Write Error
							ELSE
								udiStatus	:= fbSDOWrite.udiStatus;
							END_IF
						END_IF

					END_IF

				END_IF

			END_IF

		LifterActBGStartModOKChk:
			IF (eStatus = Idle OR eStatus = Busy) THEN

				sStatTxt	:= a_sStatText[eStat];

				bModuleOKChk	:= TRUE;
				eStatus			:= Done;

			END_IF

		LifterActBGStopModOKChk:
			IF (eStatus = Idle OR eStatus = Busy) THEN

				sStatTxt	:= a_sStatText[eStat];

				bModuleOKChk	:= FALSE;
				eStatus			:= Done;

			END_IF

		LifterActIdle:
			IF eStatus <> Idle THEN	//Reset Data
				//Private
				fbStop(bEn := FALSE);
				fbRstAxisErr(bEn := FALSE);
				fbJog(bEn := FALSE);
				fbMovRel(bEn := FALSE);
				fbMovAbs(bEn := FALSE);
				fbHoming(bEn := FALSE);
				fbPwrOff(bEn := FALSE);
				fbPwrOn(bEn := FALSE);
				fbFullHm(bEn := FALSE);
				fbFullMovAbs(bEn := FALSE);
				fbSDOWrite(bEn := FALSE);
				fbTm(IN := FALSE);
				usiStep				:= 0;
				usiCount			:= 0;
				bNotInterruptible	:= FALSE;

				sStatTxt	:= a_sStatText[eStat];

			END_IF

			eStatus	:= Idle;

			IF EDGENEG(p_bManual) THEN
				fMotionCANRstCtrlWord(ADR(tyParamOutDriver));
			END_IF

		LifterActRstNode:
			IF (eStatus = Idle OR eStatus = Busy) THEN

				eStatus	:= Busy;

				sStatTxt	:= a_sStatText[eStat];
				IF bRstErr THEN
					fbModuleOK(bEn := FALSE, bModuleOK := bModuleOK);
				END_IF
				fbModuleOK(bEn := TRUE);
				IF fbModuleOK.udiStatus = 0 THEN
					fbModuleOK(bEn := FALSE);
					eStatus			:= Done;
				ELSIF fbModuleOK.udiStatus < 65534 THEN
					eStatus		:= Error;

					IF fbModuleOK.udiStatus = 1407 THEN
						udiStatus	:= 10001;	//CANOpen Communication Error, ModuleOK Not TRUE
						fbModuleOK(bEn := FALSE);
					ELSE
						udiStatus	:= fbModuleOK.udiStatus;
					END_IF
				END_IF
			END_IF

		LifterActRstAxisErr:
			IF (eStatus = Idle OR eStatus = Busy) THEN

				eStatus	:= Busy;

				sStatTxt	:= a_sStatText[eStat];

				fbRstAxisErr(bEn := TRUE);

				IF fbRstAxisErr.udiStatus = 0 THEN
					eStatus	:= Done;
				ELSIF fbRstAxisErr.udiStatus < 65534 THEN
					udiStatus	:= fbRstAxisErr.udiStatus;
					eStatus		:= Error;
				END_IF

			END_IF

	END_CASE
END_IF

END_ACTION
```

### PullerPusher.var - Change By Project
```iecst
(*2019-04-24*)
(**)
(*Action & State & Status*)
VAR
	p_PPStat : UDINT;
	p_PPStatus : UDINT;
	p_PPStatTxt : UDINT;
END_VAR
(**)
(*Alarm*)
VAR
	p_PPAlmData : UDINT;
	p_PPAlmData1 : UDINT;
	p_PPAlmData2 : UDINT;
	p_PPAlmData3 : UDINT;
END_VAR
(**)
(*Output*)
VAR
	p_PPParamOut : UDINT;
	p_PPPwrOn : UDINT;
	p_PPIsHomed : UDINT;
	p_PPPosDiff : UDINT;
	p_PPAxisErr : UDINT;
	p_PPAxisErrID : UDINT;
	p_PPAxisErrTxt : UDINT;
	p_PPFwdLmtSen : UDINT;
	p_PPRevLmtSen : UDINT;
	p_PPActualPos : UDINT;
	p_PPWidthPosDiff : UDINT;
	p_PPJogging : UDINT;
	p_PPExtSen : UDINT;
	p_PPRetSen : UDINT;
	p_PPTurnToHm : UDINT;
END_VAR
```

### Program Logical/CANOpenServo/PullerPusher/PullerPusher (IEC) - 1.00.0 - NtMotion v5.00.0

#### InputRef.var
```iecst
(*2020-05-26*)
(**)
(*General*)
VAR
	p_eAct : REFERENCE TO ePullerPusherAction;
	p_udiRstErr : REFERENCE TO UDINT;
	p_bPrep : REFERENCE TO BOOL;
	p_bEn : REFERENCE TO BOOL;
	p_bDis : REFERENCE TO BOOL;
END_VAR
(**)
(*Configuration*)
VAR
	p_bOps : REFERENCE TO BOOL;
	p_bManual : REFERENCE TO BOOL;
	p_diWidthAtHmPos : REFERENCE TO DINT;
	p_tyTuning : REFERENCE TO tyMotionCANTuning;
	p_diGoWidth : REFERENCE TO DINT;
	p_diJogVelInUMPS : REFERENCE TO DINT;
	p_diMovePosInUM : REFERENCE TO DINT;
	p_diMoveDistInUM : REFERENCE TO DINT;
	p_diMoveVelInUMPS : REFERENCE TO DINT;
	p_diMoveAcc : REFERENCE TO DINT;
	p_diMoveDec : REFERENCE TO DINT;
	p_diMinAbsPosInUM : REFERENCE TO DINT;
	p_diMaxAbsPosInUM : REFERENCE TO DINT;
	p_diMinWidthInUM : REFERENCE TO DINT;
	p_diMaxWidthInUM : REFERENCE TO DINT;
	p_diWidthOffsetInUM : REFERENCE TO DINT;
	p_bInletSensor : REFERENCE TO BOOL;
	p_bOutletSensor : REFERENCE TO BOOL;
	p_bClearSensor : REFERENCE TO BOOL;
	p_bMiddleSensor : REFERENCE TO BOOL;
	p_bInterruptSensor : REFERENCE TO BOOL;
	p_bOpenInterruptSensor : REFERENCE TO BOOL;
	p_bCloseInterruptSensor : REFERENCE TO BOOL;
	p_bSafetyInterruptSen : REFERENCE TO BOOL;
	p_bDir : REFERENCE TO BOOL;
	p_bDirBl : REFERENCE TO BOOL;
	p_bNoIndexPulse : REFERENCE TO BOOL;
	p_usiNode : REFERENCE TO USINT;
	p_sDevice : REFERENCE TO STRING[3];
	p_sProgNm : REFERENCE TO STRING[15];
	p_diMoveBacklashDistInUM : REFERENCE TO DINT;
	p_diPitchInUM : REFERENCE TO DINT;
	p_tyParamInHm : REFERENCE TO tyMotionCANParamInHm;
	p_tyParamInConvert : REFERENCE TO tyMotionCANParamInConvert;
	p_bNtSettingsLoadDone : REFERENCE TO BOOL;
	p_bOpsAWStepMove : REFERENCE TO BOOL;
	p_eNtParamMotorType : REFERENCE TO eServoMotorType;
	p_bUITeachServo : REFERENCE TO BOOL;
	p_bOutletShutterCloseRS : REFERENCE TO BOOL;
	p_bProjInletShutPrep : REFERENCE TO BOOL;
	p_bProjOutletShutPrep : REFERENCE TO BOOL;
	p_bInletShutterCloseRS : REFERENCE TO BOOL;
	p_bInletShutterCloseRS2 : REFERENCE TO BOOL;
	p_bInletShutterCloseRS3 : REFERENCE TO BOOL;
	p_diServoTorque : REFERENCE TO DINT;
END_VAR
```

#### InputRef_Link.var
```iecst
(*2019-04-09*)
(**)
(*External Data*)
VAR
	p_bLinkOpsRun : REFERENCE TO BOOL;
	p_bLinkStartupRun : REFERENCE TO BOOL;
	p_bLinkPullConvPullerExtCtrl : REFERENCE TO BOOL;
	p_bLinkPullConvPullerRetCtrl : REFERENCE TO BOOL;
	p_bLinkDIPullerExtRS : REFERENCE TO BOOL;
	p_bLinkDIPullerRetRS : REFERENCE TO BOOL;
	p_bLinkDIPullerExtSlwRS : REFERENCE TO BOOL;
	p_bLinkDIPullerRetSlwRS : REFERENCE TO BOOL;
	p_dintLinkPullerRetSpd : REFERENCE TO DINT;
	p_dintLinkPullerRetTrq : REFERENCE TO DINT;
	p_bLinkDIPullerRotHmRS : REFERENCE TO BOOL;
END_VAR
(**)
VAR
	p_diLinkMag1TravPos : REFERENCE TO DINT;
	p_diLinkMag2TravPos : REFERENCE TO DINT;
	p_diLinkMag3TravPos : REFERENCE TO DINT;
	p_diLinkTravActualPos : REFERENCE TO DINT;
	p_bProjCurtainSenPrep : REFERENCE TO BOOL;
	p_diRcp1MtrPshrExtTorq : REFERENCE TO DINT;
	p_bMagWidthChkSen : REFERENCE TO BOOL;
	p_tyLinkTorqParam : REFERENCE TO PPTorqParam;
END_VAR
```

#### Local.var
```iecst
(*2020-05-26*)
(**)
(*Local Action, State & Status*)
VAR
	eAct : ePullerPusherAction := PPActIdle;
	eStat : ePullerPusherAction := PPActIdle;
	eMainStatus : eFBStatus := Idle;
	eStatus : eFBStatus := Idle;
	eStatus1 : eFBStatus := Idle;
	eStatus2 : eFBStatus := Idle;
	eStatus3 : eFBStatus := Idle;
	udiStatus : UDINT := 0;
	udiStatus1 : UDINT := 0;
	udiStatus2 : UDINT := 0;
	udiStatus3 : UDINT := 0;
	sStatTxt : STRING[200] := '';
	a_sStatText : ARRAY[0..50] OF STRING[200] := ['Idling','Going Width','Full Homing','Powering On','Powering Off','Homing','Moving Absolute','Moving Relative','Jogging Open','Jogging Close','Jogging Stop','Resetting Axis Error','Stopping','Writing SDO','Background Starting Module OK Check','Background Stopping Module OK Check','Going Width And Power Off','Reset Servo Module Node',33('')];
END_VAR
(**)
(*Local Alarm*)
VAR
	tyAlmData : tyAlmDat;
	tyAlmData1 : tyAlmDat;
	tyAlmData2 : tyAlmDat;
	tyAlmData3 : tyAlmDat;
	a_tyAlmText : ARRAY[10000..10299] OF tyAlmTxt := [(sAlmText:='Axis Move Abnormally By External Force',sRcyText:='Servo Motor Abnormal Operation. Reset And Resume Operation. If The Problem Persists, Please Contact Nutek For A Possible Solution.'),(sAlmText:='CANOpen Communication Error, ModuleOK Not TRUE',sRcyText:='Fail While Read/Write Data. Reset The Error And Resume Operation.'),(sAlmText:='Power On Time Out While Going New Width',sRcyText:='Timeout Expired Before Operation Completed. Reset And Resume Operation.'),(sAlmText:='Homing Time Out While Going New Width',sRcyText:='Timeout Expired Before Operation Completed. Reset And Resume Operation.'),(sAlmText:='Move Absolute Time Out While Going New Width',sRcyText:='Timeout Expired Before Operation Completed. Reset And Resume Operation.'),(sAlmText:='Stop Motion Time Out While Going New Width',sRcyText:='Timeout Expired Before Operation Completed. Reset And Resume Operation.'),(sAlmText:='Axis Error Reset Failed While Going New Width',sRcyText:='Axis Error Reset Failed. Please Retry Again Reset Operation. If The Problem Persists, Please Contact Nutek For A Possible Solution.'),(sAlmText:='Axis Error Occur In Move Absolute While Going New Width',sRcyText:='Servo Motor Abnormal Operation. Reset And Resume Operation. If The Problem Persists, Please Contact Nutek For A Possible Solution.'),(sAlmText:='Axis Error Occur In Homing While Going New Width',sRcyText:='Servo Motor Abnormal Operation. Reset And Resume Operation. If The Problem Persists, Please Contact Nutek For A Possible Solution.'),(sAlmText:='Homing Done But Home Flag Is Not Activated While Going New Width',sRcyText:='Servo Motor Abnormal Operation. Reset And Resume Operation. If The Problem Persists, Please Contact Nutek For A Possible Solution.'),(sAlmText:='Forward Limit Activated In Homing While Going New Width',sRcyText:='Forward Limit Switch Is Activated. Reset The Error By Operate The Motor Backwards.'),(sAlmText:='Reverse Limit Activated In Homing While Going New Width',sRcyText:='Reverse Limit Switch Is Activated. Reset The Error By Operate The Motor Backwards.'),(sAlmText:='Forward Limit Activated In Move Absolute While Going New Width',sRcyText:='Forward Limit Switch Is Activated. Reset The Error By Operate The Motor Backwards.'),(sAlmText:='Reverse Limit Activated In Move Absolute While Going New Width',sRcyText:='Reverse Limit Switch Is Activated. Reset The Error By Operate The Motor Backwards.'),(sAlmText:='Power On Time Out While Full Homing',sRcyText:='Timeout Expired Before Operation Completed. Reset And Resume Operation.'),(sAlmText:='Homing Time Out While Full Homing',sRcyText:='Timeout Expired Before Operation Completed. Reset And Resume Operation.'),(sAlmText:='Stop Motion Time Out While Full Homing',sRcyText:='Timeout Expired Before Operation Completed. Reset And Resume Operation.'),(sAlmText:='Axis Error Reset Failed While Full Homing',sRcyText:='Axis Error Reset Failed. Please Retry Again Reset Operation. If The Problem Persists, Please Contact Nutek For A Possible Solution.'),(sAlmText:='Axis Error Occur In Homing While Full Homing',sRcyText:='Servo Motor Abnormal Operation. Reset And Resume Operation. If The Problem Persists, Please Contact Nutek For A Possible Solution.'),(sAlmText:='Homing Done But Home Flag Is Not Activated While Full Homing',sRcyText:='Servo Motor Abnormal Operation. Reset And Resume Operation. If The Problem Persists, Please Contact Nutek For A Possible Solution.'),(sAlmText:='Forward Limit Activated In Homing While Full Homing',sRcyText:='Forward Limit Switch Is Activated. Reset The Error By Operate The Motor Backwards.'),(sAlmText:='Reverse Limit Activated In Homing While Full Homing',sRcyText:='Reverse Limit Switch Is Activated. Reset The Error By Operate The Motor Backwards.'),(sAlmText:='Power On Time Out',sRcyText:='Timeout Expired Before Operation Completed. Reset And Resume Operation.'),(sAlmText:='Power Off Time Out',sRcyText:='Timeout Expired Before Operation Completed. Reset And Resume Operation.'),(sAlmText:='Homing Time Out',sRcyText:='Timeout Expired Before Operation Completed. Reset And Resume Operation.'),(sAlmText:='Move Absolute Time Out',sRcyText:='Timeout Expired Before Operation Completed. Reset And Resume Operation.'),(sAlmText:='Move Relative Time Out',sRcyText:='Timeout Expired Before Operation Completed. Reset And Resume Operation.'),(sAlmText:='Stop Motion Time Out',sRcyText:='Timeout Expired Before Operation Completed. Reset And Resume Operation.'),(sAlmText:='SDO Write Error',sRcyText:='Fail While Write Data. Reset The Error And Resume Operation.'),(sAlmText:='Request Absolute Position Out Of Range',sRcyText:='Request Absolute Position Does Not Fall Within The Expected Range.'),(sAlmText:='Inlet Sensor Interrupt Auto Width Movement',sRcyText:='Operation Stop Due To The Interruption Of Sensor While Auto Width Moving. Solve The Interruption To Resume Operation.'),(sAlmText:='Outlet Sensor Interrupt Auto Width Movement',sRcyText:='Operation Stop Due To The Interruption Of Sensor While Auto Width Moving. Solve The Interruption To Resume Operation.'),(sAlmText:='Clear Sensor Interrupt Auto Width Movement',sRcyText:='Operation Stop Due To The Interruption Of Sensor While Auto Width Moving. Solve The Interruption To Resume Operation.'),(sAlmText:='Middle Sensor Interrupt Auto Width Movement',sRcyText:='Operation Stop Due To The Interruption Of Sensor While Auto Width Moving. Solve The Interruption To Resume Operation.'),(sAlmText:='Sensor Interrupt Auto Width Movement',sRcyText:='Operation Stop Due To The Interruption Of Sensor While Auto Width Moving. Solve The Interruption To Resume Operation.'),(sAlmText:='Power On Time Out While Going New Width And Off',sRcyText:='Timeout Expired Before Operation Completed. Reset And Resume Operation.'),(sAlmText:='Homing Time Out While Going New Width And Off',sRcyText:='Timeout Expired Before Operation Completed. Reset And Resume Operation.'),(sAlmText:='Move Absolute Time Out While Going New Width And Off',sRcyText:='Timeout Expired Before Operation Completed. Reset And Resume Operation.'),(sAlmText:='Stop Motion Time Out While Going New Width And Off',sRcyText:='Timeout Expired Before Operation Completed. Reset And Resume Operation.'),(sAlmText:='Axis Error Reset Failed While Going New Width And Off',sRcyText:='Axis Error Reset Failed. Please Retry Again Reset Operation. If The Problem Persists, Please Contact Nutek For A Possible Solution.'),(sAlmText:='Axis Error Occur In Move Absolute While Going New Width And Off',sRcyText:='Servo Motor Abnormal Operation. Reset And Resume Operation. If The Problem Persists, Please Contact Nutek For A Possible Solution.'),(sAlmText:='Axis Error Occur In Homing While Going New Width And Off',sRcyText:='Servo Motor Abnormal Operation. Reset And Resume Operation. If The Problem Persists, Please Contact Nutek For A Possible Solution.'),(sAlmText:='Homing Done But Home Flag Is Not Activated While Going New Width And Off',sRcyText:='Servo Motor Abnormal Operation. Reset And Resume Operation. If The Problem Persists, Please Contact Nutek For A Possible Solution.'),(sAlmText:='Forward Limit Activated In Homing While Going New Width And Off',sRcyText:='Forward Limit Switch Is Activated. Reset The Error By Operate The Motor Backwards.'),(sAlmText:='Reverse Limit Activated In Homing While Going New Width And Off',sRcyText:='Reverse Limit Switch Is Activated. Reset The Error By Operate The Motor Backwards.'),(sAlmText:='Forward Limit Activated In Move Absolute While Going New Width And Off',sRcyText:='Forward Limit Switch Is Activated. Reset The Error By Operate The Motor Backwards.'),(sAlmText:='Reverse Limit Activated In Move Absolute While Going New Width And Off',sRcyText:='Reverse Limit Switch Is Activated. Reset The Error By Operate The Motor Backwards.'),2((sAlmText:='Sensor Interrupt Auto Width Movement',sRcyText:='Operation Stop Due To The Interruption Of Sensor While Auto Width Moving. Solve The Interruption To Resume Operation.')),249((0)),(sAlmText:='Forward Limit Activated',sRcyText:='Forward Limit Switch Is Activated. Reset The Error By Operate The Motor Backwards.'),(sAlmText:='Reverse Limit Activated',sRcyText:='Reverse Limit Switch Is Activated. Reset The Error By Operate The Motor Backwards.')];
END_VAR
(**)
(*Local Output*)
VAR
	tyParamOut : tyMotionCANParamOut;
	sAxisErrTxt : STRING[80];
	bWidthPosDiff : BOOL;
	bJogOpen : BOOL;
	bJogClose : BOOL;
	bJogging : BOOL;
	bOpenSen : BOOL;
	bCloseSen : BOOL;
END_VAR
(**)
(*Local Input*)
VAR
	udiRstErr : UDINT := 0;
	bPrep : BOOL := TRUE;
	bEn : BOOL := TRUE;
	bDis : BOOL := FALSE;
	bOps : BOOL := FALSE;
	bManual : BOOL := FALSE;
	diWidthAtHmPos : DINT := 400;
	tyTuning : tyMotionCANTuning;
	diGoWidth : DINT := 150;
	diJogVelInUMPS : DINT := 10000;
	diMovePosInUM : DINT := 0;
	diMoveDistInUM : DINT := 0;
	diMoveVelInUMPS : DINT := 10000;
	diMoveAcc : DINT := 500;
	diMoveDec : DINT := 500;
	diMinAbsPosInUM : DINT := -3000;
	diMaxAbsPosInUM : DINT := 10000000;
	diMinWidthInUM : DINT := 70000;
	diMaxWidthInUM : DINT := 460000;
	diWidthOffsetInUM : DINT := 0;
	bInletSensor : BOOL;
	bOutletSensor : BOOL;
	bClearSensor : BOOL;
	bMiddleSensor : BOOL;
	bInterruptSensor : BOOL;
	bOpenInterruptSensor : BOOL;
	bCloseInterruptSensor : BOOL;
	bDir : BOOL;
	bDirBl : BOOL;
	bNoIndexPulse : BOOL;
	usiNode : USINT;
	sDevice : STRING[3];
	sProgNm : STRING[15] := 'AWOpen';
	diMoveBacklashDistInUM : DINT := 3000;
	diPitchInUM : DINT := 3000;
	tyParamInHm : tyMotionCANParamInHm;
	tyParamInConvert : tyMotionCANParamInConvert := (diPitchInUM:=3000);
	bNtSettingsLoadDone : BOOL := TRUE;
	eMotorType : eServoMotorType := DeltaAsdaA2;
	usiJogFwdStep : USINT;
	usiJogRevStep : USINT;
	bJogRevDone : BOOL;
	bJogFwdDone : BOOL;
	bJogStopDone : BOOL;
	bJogFwd : BOOL;
	bJogRev : BOOL;
	diServoTorque : DINT := 100;
	udiMaxTorque : UDINT := 30; (*torque value*)
	diRcp1MtrPshrExtTorq : DINT := 30; (*torque value*)
END_VAR
(**)
(*Local*)
VAR
	bRstErr : BOOL;
	udiRstErrOld : UDINT;
	bInitDone : BOOL;
	bInitialDone : BOOL;
	bModuleOKChk : BOOL := TRUE;
	bModuleOK : BOOL;
	bModuleNotOK : BOOL := TRUE;
	bModuleNotOKLock : BOOL;
	bNotInterruptible : BOOL;
	bInterruptSensor1 : BOOL;
	bInterruptSensor2 : BOOL;
	bInterruptSensor3 : BOOL;
	diActualPosInUMOld : DINT;
	usiRstStep : USINT := 0;
	usiStep : USINT;
	usiCount : USINT;
	fbTm : TON := (PT:=T#2s);
	fbServoModuleNotOk : TON := (IN:=FALSE,PT:=T#2s);
	fbServoModuleOk : TON := (IN:=FALSE,PT:=T#5s);
	fbRstNodeTimer : TON := (PT:=T#3s);
	tyParamInMove : tyMotionCANParamInMove;
	tyParamInDriver : tyMotionCANDriverIn;
	tyParamOutDriver : tyMotionCANDriverOut := (siModOfOpt_6060:=6);
	fbStop : fbMotionCANStop;
	fbRstAxisErr : fbMotionCANRstAxisErr;
	fbJog : fbMotionCANJog;
	fbMovRel : fbMotionCANMovRel;
	fbMovAbs : fbMotionCANMovAbs;
	fbHoming : fbMotionCANHoming;
	fbPwrOff : fbMotionCANPwrOff;
	fbPwrOn : fbMotionCANPwrOn;
	fbFullHm : fbMotionCANFullHm;
	fbFullMovAbs : fbMotionCANFullMovAbs;
	fbFullMovAbsBl : fbMotionCANFullMovAbsBl;
	fbModuleOK : fbMotionCANModuleOK;
	fbSDOWrite : fbCANSDOWriteArrayParam;
	fbSDOWriteTorque : CANopenSDOWrite8;
	fbPwrOnDlyTmr : TON := (PT:=T#500ms);
	bExtSlowSpd : BOOL := FALSE;
	diSlowSpeed : DINT := 4000;
	udiJogSpdAuto : UDINT := 24000;
	uiJogSpdRatio : UINT := 3000;
	usiRstJogStep : USINT;
	bRstAndExt : BOOL;
	udiModuleNum : UDINT := 301;
END_VAR
(*Output*)
VAR
	bTurnToHm : BOOL;
END_VAR
```

#### Act_Alarm2.st
```iecst
(** 2020-03-16 **)
ACTION Act_Alarm2:

	//Error
	IF EDGEPOS(eStatus2 = Error) THEN

		tyAlmData2.sProgNm		:= p_sProgNm;
		tyAlmData2.udiCode		:= udiStatus2;
		tyAlmData2.eSeverity	:= AlmSeverityError;
		tyAlmData2.udiRunTime	:= tyAlmData2.udiRunTime + 1;
		tyAlmData2.bAlm			:= TRUE;
		tyAlmData2.udiModuleNum  := udiModuleNum;
		g_sAWCloseProgNm		:= p_sProgNm;
		//Get Error Message
		IF tyAlmData2.udiCode < 10000 OR tyAlmData2.udiCode > 10099 THEN
			tyAlmData2.sAlmMsg	:= 'Unknown';
			tyAlmData2.sRcyMsg	:= 'Unknown';
		ELSE
			tyAlmData2.sAlmMsg	:= a_tyAlmText[tyAlmData2.udiCode].sAlmText;
			tyAlmData2.sRcyMsg	:= a_tyAlmText[tyAlmData2.udiCode].sRcyText;
		END_IF

		sStatTxt	:= tyAlmData2.sAlmMsg;

	ELSIF bRstErr AND (tyAlmData2.udiCode <> 0) THEN

		tyAlmData2.udiCode		:= 0;
		tyAlmData2.eSeverity	:= AlmSeverityNA;
		tyAlmData2.sAlmMsg		:= '';
		tyAlmData2.sRcyMsg		:= '';
		tyAlmData2.bAlm			:= FALSE;

		sStatTxt	:= a_sStatText[eStat];

	END_IF

END_ACTION
```
